Fanuc TP program (LS listing): 190220_hosenrohr_oV4.ls

/PROG  190220_hosenrohr_oV4
/ATTR
COMMENT	= "19-02-22 10:03:29";
PROG_SIZE	= 0;
DEFAULT_GROUP	= 1, 1, *, *, *;
/APPL
    ARC Welding Equipment: 1, *, *, *, *;
/MN
   1:  CALL HOME_ALL;
   1:  UFRAME_NUM = 1;
   1:  UTOOL_NUM = 3;
   1:  COL GUARD ADJUST 150;
   1:  ! -- Layer/Ebene 142 -- !;
   1:  PR[91] = PR[90];
   1:  PR[GP1:91,1] = PR[GP1:90,1] + -1.507;
   1:  PR[GP1:91,2] = PR[GP1:90,2] + 38.342;
   1:  PR[GP1:91,3] = PR[GP1:90,3] + 86.925;
   1:  !Sicherheitspunkt!;
   1:  PR[92] = PR[91];
   1:  PR[92] = PR[GP1:92,3] + 50;
   1:J PR[92];
   1:  !Schweissanfang anfahren!;
   1:L PR[91] R[100]mm/sec CNT100;
   1:  CALL LASER_DRAHT_START;
   1:  PR[GP1:91,1] = PR[GP1:90,1] + -7.188;
   1:  PR[GP1:91,2] = PR[GP1:90,2] + 40.092;
   1:L PR[91] R[100]mm/sec CNT100;
   1:  PR[GP1:91,1] = PR[GP1:90,1] + -15.510;
   1:  PR[GP1:91,2] = PR[GP1:90,2] + 40.391;
   1:L PR[91] R[100]mm/sec CNT100;
   1:  PR[GP1:91,1] = PR[GP1:90,1] + -22.386;
   1:  PR[GP1:91,2] = PR[GP1:90,2] + 40.265;
   1:L PR[91] R[100]mm/sec CNT100;
   1:  PR[GP1:91,1] = PR[GP1:90,1] + -29.270;
   1:  PR[GP1:91,2] = PR[GP1:90,2] + 38.008;
   1:L PR[91] R[100]mm/sec CNT100;
   1:  PR[GP1:91,1] = PR[GP1:90,1] + -36.534;
   1:  PR[GP1:91,2] = PR[GP1:90,2] + 35.327;
   1:L PR[91] R[100]mm/sec CNT100;
   1:  PR[GP1:91,1] = PR[GP1:90,1] + -41.379;
   1:  PR[GP1:91,2] = PR[GP1:90,2] + 31.493;
   1:L PR[91] R[100]mm/sec CNT100;
   1:  PR[GP1:91,1] = PR[GP1:90,1] + -47.922;
   1:  PR[GP1:91,2] = PR[GP1:90,2] + 26.092;
   1:L PR[91] R[100]mm/sec CNT100;
   1:  PR[GP1:91,1] = PR[GP1:90,1] + -50.649;
   1:  PR[GP1:91,2] = PR[GP1:90,2] + 21.582;
   1:L PR[91] R[100]mm/sec CNT100;
   1:  PR[GP1:91,1] = PR[GP1:90,1] + -55.262;
   1:  PR[GP1:91,2] = PR[GP1:90,2] + 13.777;
   1:L PR[91] R[100]mm/sec CNT100;
   1:  PR[GP1:91,1] = PR[GP1:90,1] + -56.985;
   1:  PR[GP1:91,2] = PR[GP1:90,2] + 4.269;
   1:L PR[91] R[100]mm/sec CNT100;
   1:  PR[GP1:91,1] = PR[GP1:90,1] + -57.684;
   1:  PR[GP1:91,2] = PR[GP1:90,2] + -0.066;
   1:L PR[91] R[100]mm/sec CNT100;
   1:  PR[GP1:91,1] = PR[GP1:90,1] + -56.617;
   1:  PR[GP1:91,2] = PR[GP1:90,2] + -5.926;
   1:L PR[91] R[100]mm/sec CNT100;
   1:  PR[GP1:91,1] = PR[GP1:90,1] + -56.104;
   1:  PR[GP1:91,2] = PR[GP1:90,2] + -9.354;
   1:L PR[91] R[100]mm/sec CNT100;
   1:  PR[GP1:91,1] = PR[GP1:90,1] + -55.261;
   1:  PR[GP1:91,2] = PR[GP1:90,2] + -13.923;
   1:L PR[91] R[100]mm/sec CNT100;
   1:  PR[GP1:91,1] = PR[GP1:90,1] + -50.646;
   1:  PR[GP1:91,2] = PR[GP1:90,2] + -21.730;
   1:L PR[91] R[100]mm/sec CNT100;
   1:  PR[GP1:91,1] = PR[GP1:90,1] + -47.919;
   1:  PR[GP1:91,2] = PR[GP1:90,2] + -26.240;
   1:L PR[91] R[100]mm/sec CNT100;
   1:  PR[GP1:91,1] = PR[GP1:90,1] + -41.373;
   1:  PR[GP1:91,2] = PR[GP1:90,2] + -31.640;
   1:L PR[91] R[100]mm/sec CNT100;
   1:  PR[GP1:91,1] = PR[GP1:90,1] + -36.528;
   1:  PR[GP1:91,2] = PR[GP1:90,2] + -35.474;
   1:L PR[91] R[100]mm/sec CNT100;
   1:  PR[GP1:91,1] = PR[GP1:90,1] + -29.263;
   1:  PR[GP1:91,2] = PR[GP1:90,2] + -38.152;
   1:L PR[91] R[100]mm/sec CNT100;
   1:  PR[GP1:91,1] = PR[GP1:90,1] + -22.379;
   1:  PR[GP1:91,2] = PR[GP1:90,2] + -40.411;
   1:L PR[91] R[100]mm/sec CNT100;
   1:  PR[GP1:91,1] = PR[GP1:90,1] + -15.502;
   1:  PR[GP1:91,2] = PR[GP1:90,2] + -40.533;
   1:L PR[91] R[100]mm/sec CNT100;
   1:  PR[GP1:91,1] = PR[GP1:90,1] + -7.183;
   1:  PR[GP1:91,2] = PR[GP1:90,2] + -40.236;
   1:L PR[91] R[100]mm/sec CNT100;
   1:  PR[GP1:91,1] = PR[GP1:90,1] + -1.509;
   1:  PR[GP1:91,2] = PR[GP1:90,2] + -38.475;
   1:L PR[91] R[100]mm/sec CNT100;
   1:  PR[GP1:91,1] = PR[GP1:90,1] + 1.722;
   1:  PR[GP1:91,2] = PR[GP1:90,2] + -38.474;
   1:L PR[91] R[100]mm/sec CNT100;
   1:  PR[GP1:91,1] = PR[GP1:90,1] + 7.396;
   1:  PR[GP1:91,2] = PR[GP1:90,2] + -40.236;
   1:L PR[91] R[100]mm/sec CNT100;
   1:  PR[GP1:91,1] = PR[GP1:90,1] + 15.715;
   1:  PR[GP1:91,2] = PR[GP1:90,2] + -40.532;
   1:L PR[91] R[100]mm/sec CNT100;
   1:  PR[GP1:91,1] = PR[GP1:90,1] + 22.592;
   1:  PR[GP1:91,2] = PR[GP1:90,2] + -40.411;
   1:L PR[91] R[100]mm/sec CNT100;
   1:  PR[GP1:91,1] = PR[GP1:90,1] + 29.475;
   1:  PR[GP1:91,2] = PR[GP1:90,2] + -38.153;
   1:L PR[91] R[100]mm/sec CNT100;
   1:  PR[GP1:91,1] = PR[GP1:90,1] + 36.742;
   1:  PR[GP1:91,2] = PR[GP1:90,2] + -35.476;
   1:L PR[91] R[100]mm/sec CNT100;
   1:  PR[GP1:91,1] = PR[GP1:90,1] + 41.585;
   1:  PR[GP1:91,2] = PR[GP1:90,2] + -31.641;
   1:L PR[91] R[100]mm/sec CNT100;
   1:  PR[GP1:91,1] = PR[GP1:90,1] + 48.132;
   1:  PR[GP1:91,2] = PR[GP1:90,2] + -26.235;
   1:L PR[91] R[100]mm/sec CNT100;
   1:  PR[GP1:91,1] = PR[GP1:90,1] + 50.859;
   1:  PR[GP1:91,2] = PR[GP1:90,2] + -21.727;
   1:L PR[91] R[100]mm/sec CNT100;
   1:  PR[GP1:91,1] = PR[GP1:90,1] + 55.474;
   1:  PR[GP1:91,2] = PR[GP1:90,2] + -13.938;
   1:L PR[91] R[100]mm/sec CNT100;
   1:  PR[GP1:91,1] = PR[GP1:90,1] + 57.199;
   1:  PR[GP1:91,2] = PR[GP1:90,2] + -4.414;
   1:L PR[91] R[100]mm/sec CNT100;
   1:  PR[GP1:91,1] = PR[GP1:90,1] + 57.897;
   1:  PR[GP1:91,2] = PR[GP1:90,2] + -0.078;
   1:L PR[91] R[100]mm/sec CNT100;
   1:  PR[GP1:91,1] = PR[GP1:90,1] + 56.831;
   1:  PR[GP1:91,2] = PR[GP1:90,2] + 5.789;
   1:L PR[91] R[100]mm/sec CNT100;
   1:  PR[GP1:91,1] = PR[GP1:90,1] + 56.318;
   1:  PR[GP1:91,2] = PR[GP1:90,2] + 9.220;
   1:L PR[91] R[100]mm/sec CNT100;
   1:  PR[GP1:91,1] = PR[GP1:90,1] + 55.475;
   1:  PR[GP1:91,2] = PR[GP1:90,2] + 13.790;
   1:L PR[91] R[100]mm/sec CNT100;
   1:  PR[GP1:91,1] = PR[GP1:90,1] + 50.862;
   1:  PR[GP1:91,2] = PR[GP1:90,2] + 21.580;
   1:L PR[91] R[100]mm/sec CNT100;
   1:  PR[GP1:91,1] = PR[GP1:90,1] + 48.135;
   1:  PR[GP1:91,2] = PR[GP1:90,2] + 26.088;
   1:L PR[91] R[100]mm/sec CNT100;
   1:  PR[GP1:91,1] = PR[GP1:90,1] + 41.591;
   1:  PR[GP1:91,2] = PR[GP1:90,2] + 31.494;
   1:L PR[91] R[100]mm/sec CNT100;
   1:  PR[GP1:91,1] = PR[GP1:90,1] + 36.747;
   1:  PR[GP1:91,2] = PR[GP1:90,2] + 35.329;
   1:L PR[91] R[100]mm/sec CNT100;
   1:  PR[GP1:91,1] = PR[GP1:90,1] + 29.483;
   1:  PR[GP1:91,2] = PR[GP1:90,2] + 38.008;
   1:L PR[91] R[100]mm/sec CNT100;
   1:  PR[GP1:91,1] = PR[GP1:90,1] + 22.599;
   1:  PR[GP1:91,2] = PR[GP1:90,2] + 40.266;
   1:L PR[91] R[100]mm/sec CNT100;
   1:  PR[GP1:91,1] = PR[GP1:90,1] + 15.722;
   1:  PR[GP1:91,2] = PR[GP1:90,2] + 40.390;
   1:L PR[91] R[100]mm/sec CNT100;
   1:  PR[GP1:91,1] = PR[GP1:90,1] + 7.401;
   1:  PR[GP1:91,2] = PR[GP1:90,2] + 40.092;
   1:L PR[91] R[100]mm/sec CNT100;
   1:  PR[GP1:91,1] = PR[GP1:90,1] + 1.720;
   1:  PR[GP1:91,2] = PR[GP1:90,2] + 38.342;
   1:L PR[91] R[100]mm/sec CNT100;
   1:  ! -- Layer/Ebene 143 -- !;
   1:  PR[91] = PR[90];
   1:  PR[GP1:91,1] = PR[GP1:90,1] + -1.481;
   1:  PR[GP1:91,2] = PR[GP1:90,2] + 38.516;
   1:  PR[GP1:91,3] = PR[GP1:90,3] + 87.535;
   1:L PR[91] R[100]mm/sec CNT100;
   1:  PR[GP1:91,1] = PR[GP1:90,1] + -6.890;
   1:  PR[GP1:91,2] = PR[GP1:90,2] + 40.181;
   1:L PR[91] R[100]mm/sec CNT100;
   1:  PR[GP1:91,1] = PR[GP1:90,1] + -15.548;
   1:  PR[GP1:91,2] = PR[GP1:90,2] + 40.491;
   1:L PR[91] R[100]mm/sec CNT100;
   1:  PR[GP1:91,1] = PR[GP1:90,1] + -22.125;
   1:  PR[GP1:91,2] = PR[GP1:90,2] + 40.371;
   1:L PR[91] R[100]mm/sec CNT100;
   1:  PR[GP1:91,1] = PR[GP1:90,1] + -29.339;
   1:  PR[GP1:91,2] = PR[GP1:90,2] + 38.006;
   1:L PR[91] R[100]mm/sec CNT100;
   1:  PR[GP1:91,1] = PR[GP1:90,1] + -36.313;
   1:  PR[GP1:91,2] = PR[GP1:90,2] + 35.432;
   1:L PR[91] R[100]mm/sec CNT100;
   1:  PR[GP1:91,1] = PR[GP1:90,1] + -41.439;
   1:  PR[GP1:91,2] = PR[GP1:90,2] + 31.376;
   1:L PR[91] R[100]mm/sec CNT100;
   1:  PR[GP1:91,1] = PR[GP1:90,1] + -47.738;
   1:  PR[GP1:91,2] = PR[GP1:90,2] + 26.177;
   1:L PR[91] R[100]mm/sec CNT100;
   1:  PR[GP1:91,1] = PR[GP1:90,1] + -50.656;
   1:  PR[GP1:91,2] = PR[GP1:90,2] + 21.350;
   1:L PR[91] R[100]mm/sec CNT100;
   1:  PR[GP1:91,1] = PR[GP1:90,1] + -55.103;
   1:  PR[GP1:91,2] = PR[GP1:90,2] + 13.825;
   1:L PR[91] R[100]mm/sec CNT100;
   1:  PR[GP1:91,1] = PR[GP1:90,1] + -56.765;
   1:  PR[GP1:91,2] = PR[GP1:90,2] + 4.657;
   1:L PR[91] R[100]mm/sec CNT100;
   1:  PR[GP1:91,1] = PR[GP1:90,1] + -57.526;
   1:  PR[GP1:91,2] = PR[GP1:90,2] + -0.066;
   1:L PR[91] R[100]mm/sec CNT100;
   1:  PR[GP1:91,1] = PR[GP1:90,1] + -56.569;
   1:  PR[GP1:91,2] = PR[GP1:90,2] + -5.328;
   1:L PR[91] R[100]mm/sec CNT100;
   1:  PR[GP1:91,1] = PR[GP1:90,1] + -56.014;
   1:  PR[GP1:91,2] = PR[GP1:90,2] + -9.028;
   1:L PR[91] R[100]mm/sec CNT100;
   1:  PR[GP1:91,1] = PR[GP1:90,1] + -55.103;
   1:  PR[GP1:91,2] = PR[GP1:90,2] + -13.970;
   1:L PR[91] R[100]mm/sec CNT100;
   1:  PR[GP1:91,1] = PR[GP1:90,1] + -50.653;
   1:  PR[GP1:91,2] = PR[GP1:90,2] + -21.498;
   1:L PR[91] R[100]mm/sec CNT100;
   1:  PR[GP1:91,1] = PR[GP1:90,1] + -47.735;
   1:  PR[GP1:91,2] = PR[GP1:90,2] + -26.324;
   1:L PR[91] R[100]mm/sec CNT100;
   1:  PR[GP1:91,1] = PR[GP1:90,1] + -41.433;
   1:  PR[GP1:91,2] = PR[GP1:90,2] + -31.523;
   1:L PR[91] R[100]mm/sec CNT100;
   1:  PR[GP1:91,1] = PR[GP1:90,1] + -36.307;
   1:  PR[GP1:91,2] = PR[GP1:90,2] + -35.579;
   1:L PR[91] R[100]mm/sec CNT100;
   1:  PR[GP1:91,1] = PR[GP1:90,1] + -29.332;
   1:  PR[GP1:91,2] = PR[GP1:90,2] + -38.150;
   1:L PR[91] R[100]mm/sec CNT100;
   1:  PR[GP1:91,1] = PR[GP1:90,1] + -22.118;
   1:  PR[GP1:91,2] = PR[GP1:90,2] + -40.517;
   1:L PR[91] R[100]mm/sec CNT100;
   1:  PR[GP1:91,1] = PR[GP1:90,1] + -15.540;
   1:  PR[GP1:91,2] = PR[GP1:90,2] + -40.633;
   1:L PR[91] R[100]mm/sec CNT100;
   1:  PR[GP1:91,1] = PR[GP1:90,1] + -6.886;
   1:  PR[GP1:91,2] = PR[GP1:90,2] + -40.325;
   1:L PR[91] R[100]mm/sec CNT100;
   1:  PR[GP1:91,1] = PR[GP1:90,1] + -1.483;
   1:  PR[GP1:91,2] = PR[GP1:90,2] + -38.649;
   1:L PR[91] R[100]mm/sec CNT100;
   1:  PR[GP1:91,1] = PR[GP1:90,1] + 1.697;
   1:  PR[GP1:91,2] = PR[GP1:90,2] + -38.648;
   1:L PR[91] R[100]mm/sec CNT100;
   1:  PR[GP1:91,1] = PR[GP1:90,1] + 7.100;
   1:  PR[GP1:91,2] = PR[GP1:90,2] + -40.325;
   1:L PR[91] R[100]mm/sec CNT100;
   1:  PR[GP1:91,1] = PR[GP1:90,1] + 15.753;
   1:  PR[GP1:91,2] = PR[GP1:90,2] + -40.633;
   1:L PR[91] R[100]mm/sec CNT100;
   1:  PR[GP1:91,1] = PR[GP1:90,1] + 22.331;
   1:  PR[GP1:91,2] = PR[GP1:90,2] + -40.517;
   1:L PR[91] R[100]mm/sec CNT100;
   1:  PR[GP1:91,1] = PR[GP1:90,1] + 29.544;
   1:  PR[GP1:91,2] = PR[GP1:90,2] + -38.150;
   1:L PR[91] R[100]mm/sec CNT100;
   1:  PR[GP1:91,1] = PR[GP1:90,1] + 36.520;
   1:  PR[GP1:91,2] = PR[GP1:90,2] + -35.581;
   1:L PR[91] R[100]mm/sec CNT100;
   1:  PR[GP1:91,1] = PR[GP1:90,1] + 41.646;
   1:  PR[GP1:91,2] = PR[GP1:90,2] + -31.523;
   1:L PR[91] R[100]mm/sec CNT100;
   1:  PR[GP1:91,1] = PR[GP1:90,1] + 47.948;
   1:  PR[GP1:91,2] = PR[GP1:90,2] + -26.319;
   1:L PR[91] R[100]mm/sec CNT100;
   1:  PR[GP1:91,1] = PR[GP1:90,1] + 50.866;
   1:  PR[GP1:91,2] = PR[GP1:90,2] + -21.495;
   1:L PR[91] R[100]mm/sec CNT100;
   1:  PR[GP1:91,1] = PR[GP1:90,1] + 55.315;
   1:  PR[GP1:91,2] = PR[GP1:90,2] + -13.984;
   1:L PR[91] R[100]mm/sec CNT100;
   1:  PR[GP1:91,1] = PR[GP1:90,1] + 56.979;
   1:  PR[GP1:91,2] = PR[GP1:90,2] + -4.802;
   1:L PR[91] R[100]mm/sec CNT100;
   1:  PR[GP1:91,1] = PR[GP1:90,1] + 57.740;
   1:  PR[GP1:91,2] = PR[GP1:90,2] + -0.078;
   1:L PR[91] R[100]mm/sec CNT100;
   1:  PR[GP1:91,1] = PR[GP1:90,1] + 56.782;
   1:  PR[GP1:91,2] = PR[GP1:90,2] + 5.190;
   1:L PR[91] R[100]mm/sec CNT100;
   1:  PR[GP1:91,1] = PR[GP1:90,1] + 56.228;
   1:  PR[GP1:91,2] = PR[GP1:90,2] + 8.895;
   1:L PR[91] R[100]mm/sec CNT100;
   1:  PR[GP1:91,1] = PR[GP1:90,1] + 55.317;
   1:  PR[GP1:91,2] = PR[GP1:90,2] + 13.837;
   1:L PR[91] R[100]mm/sec CNT100;
   1:  PR[GP1:91,1] = PR[GP1:90,1] + 50.869;
   1:  PR[GP1:91,2] = PR[GP1:90,2] + 21.347;
   1:L PR[91] R[100]mm/sec CNT100;
   1:  PR[GP1:91,1] = PR[GP1:90,1] + 47.951;
   1:  PR[GP1:91,2] = PR[GP1:90,2] + 26.172;
   1:L PR[91] R[100]mm/sec CNT100;
   1:  PR[GP1:91,1] = PR[GP1:90,1] + 41.651;
   1:  PR[GP1:91,2] = PR[GP1:90,2] + 31.377;
   1:L PR[91] R[100]mm/sec CNT100;
   1:  PR[GP1:91,1] = PR[GP1:90,1] + 36.526;
   1:  PR[GP1:91,2] = PR[GP1:90,2] + 35.434;
   1:L PR[91] R[100]mm/sec CNT100;
   1:  PR[GP1:91,1] = PR[GP1:90,1] + 29.552;
   1:  PR[GP1:91,2] = PR[GP1:90,2] + 38.006;
   1:L PR[91] R[100]mm/sec CNT100;
   1:  PR[GP1:91,1] = PR[GP1:90,1] + 22.338;
   1:  PR[GP1:91,2] = PR[GP1:90,2] + 40.372;
   1:L PR[91] R[100]mm/sec CNT100;
   1:  PR[GP1:91,1] = PR[GP1:90,1] + 15.761;
   1:  PR[GP1:91,2] = PR[GP1:90,2] + 40.491;
   1:L PR[91] R[100]mm/sec CNT100;
   1:  PR[GP1:91,1] = PR[GP1:90,1] + 7.103;
   1:  PR[GP1:91,2] = PR[GP1:90,2] + 40.181;
   1:L PR[91] R[100]mm/sec CNT100;
   1:  PR[GP1:91,1] = PR[GP1:90,1] + 1.695;
   1:  PR[GP1:91,2] = PR[GP1:90,2] + 38.515;
   1:L PR[91] R[100]mm/sec CNT100;
   1:  ! -- Layer/Ebene 144 -- !;
   1:  PR[91] = PR[90];
   1:  PR[GP1:91,1] = PR[GP1:90,1] + -1.456;
   1:  PR[GP1:91,2] = PR[GP1:90,2] + 38.689;
   1:  PR[GP1:91,3] = PR[GP1:90,3] + 88.145;
   1:L PR[91] R[100]mm/sec CNT100;
   1:  PR[GP1:91,1] = PR[GP1:90,1] + -6.592;
   1:  PR[GP1:91,2] = PR[GP1:90,2] + 40.270;
   1:L PR[91] R[100]mm/sec CNT100;
   1:  PR[GP1:91,1] = PR[GP1:90,1] + -15.586;
   1:  PR[GP1:91,2] = PR[GP1:90,2] + 40.592;
   1:L PR[91] R[100]mm/sec CNT100;
   1:  PR[GP1:91,1] = PR[GP1:90,1] + -21.864;
   1:  PR[GP1:91,2] = PR[GP1:90,2] + 40.477;
   1:L PR[91] R[100]mm/sec CNT100;
   1:  PR[GP1:91,1] = PR[GP1:90,1] + -29.408;
   1:  PR[GP1:91,2] = PR[GP1:90,2] + 38.003;
   1:L PR[91] R[100]mm/sec CNT100;
   1:  PR[GP1:91,1] = PR[GP1:90,1] + -36.091;
   1:  PR[GP1:91,2] = PR[GP1:90,2] + 35.537;
   1:L PR[91] R[100]mm/sec CNT100;
   1:  PR[GP1:91,1] = PR[GP1:90,1] + -41.499;
   1:  PR[GP1:91,2] = PR[GP1:90,2] + 31.258;
   1:L PR[91] R[100]mm/sec CNT100;
   1:  PR[GP1:91,1] = PR[GP1:90,1] + -47.553;
   1:  PR[GP1:91,2] = PR[GP1:90,2] + 26.261;
   1:L PR[91] R[100]mm/sec CNT100;
   1:  PR[GP1:91,1] = PR[GP1:90,1] + -50.663;
   1:  PR[GP1:91,2] = PR[GP1:90,2] + 21.117;
   1:L PR[91] R[100]mm/sec CNT100;
   1:  PR[GP1:91,1] = PR[GP1:90,1] + -54.945;
   1:  PR[GP1:91,2] = PR[GP1:90,2] + 13.872;
   1:L PR[91] R[100]mm/sec CNT100;
   1:  PR[GP1:91,1] = PR[GP1:90,1] + -56.545;
   1:  PR[GP1:91,2] = PR[GP1:90,2] + 5.045;
   1:L PR[91] R[100]mm/sec CNT100;
   1:  PR[GP1:91,1] = PR[GP1:90,1] + -57.369;
   1:  PR[GP1:91,2] = PR[GP1:90,2] + -0.066;
   1:L PR[91] R[100]mm/sec CNT100;
   1:  PR[GP1:91,1] = PR[GP1:90,1] + -56.520;
   1:  PR[GP1:91,2] = PR[GP1:90,2] + -4.730;
   1:L PR[91] R[100]mm/sec CNT100;
   1:  PR[GP1:91,1] = PR[GP1:90,1] + -55.925;
   1:  PR[GP1:91,2] = PR[GP1:90,2] + -8.703;
   1:L PR[91] R[100]mm/sec CNT100;
   1:  PR[GP1:91,1] = PR[GP1:90,1] + -54.944;
   1:  PR[GP1:91,2] = PR[GP1:90,2] + -14.017;
   1:L PR[91] R[100]mm/sec CNT100;
   1:  PR[GP1:91,1] = PR[GP1:90,1] + -50.660;
   1:  PR[GP1:91,2] = PR[GP1:90,2] + -21.265;
   1:L PR[91] R[100]mm/sec CNT100;
   1:  PR[GP1:91,1] = PR[GP1:90,1] + -47.550;
   1:  PR[GP1:91,2] = PR[GP1:90,2] + -26.408;
   1:L PR[91] R[100]mm/sec CNT100;
   1:  PR[GP1:91,1] = PR[GP1:90,1] + -41.493;
   1:  PR[GP1:91,2] = PR[GP1:90,2] + -31.405;
   1:L PR[91] R[100]mm/sec CNT100;
   1:  PR[GP1:91,1] = PR[GP1:90,1] + -36.086;
   1:  PR[GP1:91,2] = PR[GP1:90,2] + -35.684;
   1:L PR[91] R[100]mm/sec CNT100;
   1:  PR[GP1:91,1] = PR[GP1:90,1] + -29.401;
   1:  PR[GP1:91,2] = PR[GP1:90,2] + -38.148;
   1:L PR[91] R[100]mm/sec CNT100;
   1:  PR[GP1:91,1] = PR[GP1:90,1] + -21.857;
   1:  PR[GP1:91,2] = PR[GP1:90,2] + -40.623;
   1:L PR[91] R[100]mm/sec CNT100;
   1:  PR[GP1:91,1] = PR[GP1:90,1] + -15.579;
   1:  PR[GP1:91,2] = PR[GP1:90,2] + -40.734;
   1:L PR[91] R[100]mm/sec CNT100;
   1:  PR[GP1:91,1] = PR[GP1:90,1] + -6.589;
   1:  PR[GP1:91,2] = PR[GP1:90,2] + -40.414;
   1:L PR[91] R[100]mm/sec CNT100;
   1:  PR[GP1:91,1] = PR[GP1:90,1] + -1.458;
   1:  PR[GP1:91,2] = PR[GP1:90,2] + -38.822;
   1:L PR[91] R[100]mm/sec CNT100;
   1:  PR[GP1:91,1] = PR[GP1:90,1] + 1.671;
   1:L PR[91] R[100]mm/sec CNT100;
   1:  PR[GP1:91,1] = PR[GP1:90,1] + 6.803;
   1:  PR[GP1:91,2] = PR[GP1:90,2] + -40.413;
   1:L PR[91] R[100]mm/sec CNT100;
   1:  PR[GP1:91,1] = PR[GP1:90,1] + 15.792;
   1:  PR[GP1:91,2] = PR[GP1:90,2] + -40.734;
   1:L PR[91] R[100]mm/sec CNT100;
   1:  PR[GP1:91,1] = PR[GP1:90,1] + 22.071;
   1:  PR[GP1:91,2] = PR[GP1:90,2] + -40.623;
   1:L PR[91] R[100]mm/sec CNT100;
   1:  PR[GP1:91,1] = PR[GP1:90,1] + 29.613;
   1:  PR[GP1:91,2] = PR[GP1:90,2] + -38.148;
   1:L PR[91] R[100]mm/sec CNT100;
   1:  PR[GP1:91,1] = PR[GP1:90,1] + 36.299;
   1:  PR[GP1:91,2] = PR[GP1:90,2] + -35.685;
   1:L PR[91] R[100]mm/sec CNT100;
   1:  PR[GP1:91,1] = PR[GP1:90,1] + 41.706;
   1:  PR[GP1:91,2] = PR[GP1:90,2] + -31.405;
   1:L PR[91] R[100]mm/sec CNT100;
   1:  PR[GP1:91,1] = PR[GP1:90,1] + 47.763;
   1:  PR[GP1:91,2] = PR[GP1:90,2] + -26.403;
   1:L PR[91] R[100]mm/sec CNT100;
   1:  PR[GP1:91,1] = PR[GP1:90,1] + 50.873;
   1:  PR[GP1:91,2] = PR[GP1:90,2] + -21.262;
   1:L PR[91] R[100]mm/sec CNT100;
   1:  PR[GP1:91,1] = PR[GP1:90,1] + 55.157;
   1:  PR[GP1:91,2] = PR[GP1:90,2] + -14.031;
   1:L PR[91] R[100]mm/sec CNT100;
   1:  PR[GP1:91,1] = PR[GP1:90,1] + 56.758;
   1:  PR[GP1:91,2] = PR[GP1:90,2] + -5.190;
   1:L PR[91] R[100]mm/sec CNT100;
   1:  PR[GP1:91,1] = PR[GP1:90,1] + 57.582;
   1:  PR[GP1:91,2] = PR[GP1:90,2] + -0.078;
   1:L PR[91] R[100]mm/sec CNT100;
   1:  PR[GP1:91,1] = PR[GP1:90,1] + 56.733;
   1:  PR[GP1:91,2] = PR[GP1:90,2] + 4.591;
   1:L PR[91] R[100]mm/sec CNT100;
   1:  PR[GP1:91,1] = PR[GP1:90,1] + 56.139;
   1:  PR[GP1:91,2] = PR[GP1:90,2] + 8.569;
   1:L PR[91] R[100]mm/sec CNT100;
   1:  PR[GP1:91,1] = PR[GP1:90,1] + 55.158;
   1:  PR[GP1:91,2] = PR[GP1:90,2] + 13.884;
   1:L PR[91] R[100]mm/sec CNT100;
   1:  PR[GP1:91,1] = PR[GP1:90,1] + 50.876;
   1:  PR[GP1:91,2] = PR[GP1:90,2] + 21.115;
   1:L PR[91] R[100]mm/sec CNT100;
   1:  PR[GP1:91,1] = PR[GP1:90,1] + 47.766;
   1:  PR[GP1:91,2] = PR[GP1:90,2] + 26.256;
   1:L PR[91] R[100]mm/sec CNT100;
   1:  PR[GP1:91,1] = PR[GP1:90,1] + 41.711;
   1:  PR[GP1:91,2] = PR[GP1:90,2] + 31.259;
   1:L PR[91] R[100]mm/sec CNT100;
   1:  PR[GP1:91,1] = PR[GP1:90,1] + 36.304;
   1:  PR[GP1:91,2] = PR[GP1:90,2] + 35.539;
   1:L PR[91] R[100]mm/sec CNT100;
   1:  PR[GP1:91,1] = PR[GP1:90,1] + 29.620;
   1:  PR[GP1:91,2] = PR[GP1:90,2] + 38.004;
   1:L PR[91] R[100]mm/sec CNT100;
   1:  PR[GP1:91,1] = PR[GP1:90,1] + 22.077;
   1:  PR[GP1:91,2] = PR[GP1:90,2] + 40.478;
   1:L PR[91] R[100]mm/sec CNT100;
   1:  PR[GP1:91,1] = PR[GP1:90,1] + 15.799;
   1:  PR[GP1:91,2] = PR[GP1:90,2] + 40.591;
   1:L PR[91] R[100]mm/sec CNT100;
   1:  PR[GP1:91,1] = PR[GP1:90,1] + 6.806;
   1:  PR[GP1:91,2] = PR[GP1:90,2] + 40.269;
   1:L PR[91] R[100]mm/sec CNT100;
   1:  PR[GP1:91,1] = PR[GP1:90,1] + 1.670;
   1:  PR[GP1:91,2] = PR[GP1:90,2] + 38.688;
   1:L PR[91] R[100]mm/sec CNT100;
   1:  ! -- Layer/Ebene 145 -- !;
   1:  PR[91] = PR[90];
   1:  PR[GP1:91,1] = PR[GP1:90,1] + -1.431;
   1:  PR[GP1:91,2] = PR[GP1:90,2] + 38.862;
   1:  PR[GP1:91,3] = PR[GP1:90,3] + 88.755;
   1:L PR[91] R[100]mm/sec CNT100;
   1:  PR[GP1:91,1] = PR[GP1:90,1] + -6.295;
   1:  PR[GP1:91,2] = PR[GP1:90,2] + 40.358;
   1:L PR[91] R[100]mm/sec CNT100;
   1:  PR[GP1:91,1] = PR[GP1:90,1] + -15.624;
   1:  PR[GP1:91,2] = PR[GP1:90,2] + 40.693;
   1:L PR[91] R[100]mm/sec CNT100;
   1:  PR[GP1:91,1] = PR[GP1:90,1] + -21.602;
   1:  PR[GP1:91,2] = PR[GP1:90,2] + 40.584;
   1:L PR[91] R[100]mm/sec CNT100;
   1:  PR[GP1:91,1] = PR[GP1:90,1] + -29.476;
   1:  PR[GP1:91,2] = PR[GP1:90,2] + 38.002;
   1:L PR[91] R[100]mm/sec CNT100;
   1:  PR[GP1:91,1] = PR[GP1:90,1] + -35.870;
   1:  PR[GP1:91,2] = PR[GP1:90,2] + 35.642;
   1:L PR[91] R[100]mm/sec CNT100;
   1:  PR[GP1:91,1] = PR[GP1:90,1] + -41.558;
   1:  PR[GP1:91,2] = PR[GP1:90,2] + 31.140;
   1:L PR[91] R[100]mm/sec CNT100;
   1:  PR[GP1:91,1] = PR[GP1:90,1] + -47.368;
   1:  PR[GP1:91,2] = PR[GP1:90,2] + 26.345;
   1:L PR[91] R[100]mm/sec CNT100;
   1:  PR[GP1:91,1] = PR[GP1:90,1] + -50.670;
   1:  PR[GP1:91,2] = PR[GP1:90,2] + 20.884;
   1:L PR[91] R[100]mm/sec CNT100;
   1:  PR[GP1:91,1] = PR[GP1:90,1] + -54.786;
   1:  PR[GP1:91,2] = PR[GP1:90,2] + 13.919;
   1:L PR[91] R[100]mm/sec CNT100;
   1:  PR[GP1:91,1] = PR[GP1:90,1] + -56.324;
   1:  PR[GP1:91,2] = PR[GP1:90,2] + 5.433;
   1:L PR[91] R[100]mm/sec CNT100;
   1:  PR[GP1:91,1] = PR[GP1:90,1] + -57.211;
   1:  PR[GP1:91,2] = PR[GP1:90,2] + -0.066;
   1:L PR[91] R[100]mm/sec CNT100;
   1:  PR[GP1:91,1] = PR[GP1:90,1] + -56.471;
   1:  PR[GP1:91,2] = PR[GP1:90,2] + -4.131;
   1:L PR[91] R[100]mm/sec CNT100;
   1:  PR[GP1:91,1] = PR[GP1:90,1] + -55.835;
   1:  PR[GP1:91,2] = PR[GP1:90,2] + -8.377;
   1:L PR[91] R[100]mm/sec CNT100;
   1:  PR[GP1:91,1] = PR[GP1:90,1] + -54.786;
   1:  PR[GP1:91,2] = PR[GP1:90,2] + -14.064;
   1:L PR[91] R[100]mm/sec CNT100;
   1:  PR[GP1:91,1] = PR[GP1:90,1] + -50.667;
   1:  PR[GP1:91,2] = PR[GP1:90,2] + -21.032;
   1:L PR[91] R[100]mm/sec CNT100;
   1:  PR[GP1:91,1] = PR[GP1:90,1] + -47.366;
   1:  PR[GP1:91,2] = PR[GP1:90,2] + -26.492;
   1:L PR[91] R[100]mm/sec CNT100;
   1:  PR[GP1:91,1] = PR[GP1:90,1] + -41.553;
   1:  PR[GP1:91,2] = PR[GP1:90,2] + -31.287;
   1:L PR[91] R[100]mm/sec CNT100;
   1:  PR[GP1:91,1] = PR[GP1:90,1] + -35.865;
   1:  PR[GP1:91,2] = PR[GP1:90,2] + -35.789;
   1:L PR[91] R[100]mm/sec CNT100;
   1:  PR[GP1:91,1] = PR[GP1:90,1] + -29.469;
   1:  PR[GP1:91,2] = PR[GP1:90,2] + -38.146;
   1:L PR[91] R[100]mm/sec CNT100;
   1:  PR[GP1:91,1] = PR[GP1:90,1] + -21.596;
   1:  PR[GP1:91,2] = PR[GP1:90,2] + -40.729;
   1:L PR[91] R[100]mm/sec CNT100;
   1:  PR[GP1:91,1] = PR[GP1:90,1] + -15.618;
   1:  PR[GP1:91,2] = PR[GP1:90,2] + -40.835;
   1:L PR[91] R[100]mm/sec CNT100;
   1:  PR[GP1:91,1] = PR[GP1:90,1] + -6.292;
   1:  PR[GP1:91,2] = PR[GP1:90,2] + -40.502;
   1:L PR[91] R[100]mm/sec CNT100;
   1:  PR[GP1:91,1] = PR[GP1:90,1] + -1.433;
   1:  PR[GP1:91,2] = PR[GP1:90,2] + -38.996;
   1:L PR[91] R[100]mm/sec CNT100;
   1:  PR[GP1:91,1] = PR[GP1:90,1] + 1.646;
   1:  PR[GP1:91,2] = PR[GP1:90,2] + -38.995;
   1:L PR[91] R[100]mm/sec CNT100;
   1:  PR[GP1:91,1] = PR[GP1:90,1] + 6.506;
   1:  PR[GP1:91,2] = PR[GP1:90,2] + -40.502;
   1:L PR[91] R[100]mm/sec CNT100;
   1:  PR[GP1:91,1] = PR[GP1:90,1] + 15.831;
   1:  PR[GP1:91,2] = PR[GP1:90,2] + -40.834;
   1:L PR[91] R[100]mm/sec CNT100;
   1:  PR[GP1:91,1] = PR[GP1:90,1] + 21.810;
   1:  PR[GP1:91,2] = PR[GP1:90,2] + -40.729;
   1:L PR[91] R[100]mm/sec CNT100;
   1:  PR[GP1:91,1] = PR[GP1:90,1] + 29.682;
   1:  PR[GP1:91,2] = PR[GP1:90,2] + -38.146;
   1:L PR[91] R[100]mm/sec CNT100;
   1:  PR[GP1:91,1] = PR[GP1:90,1] + 36.078;
   1:  PR[GP1:91,2] = PR[GP1:90,2] + -35.790;
   1:L PR[91] R[100]mm/sec CNT100;
   1:  PR[GP1:91,1] = PR[GP1:90,1] + 41.766;
   1:  PR[GP1:91,2] = PR[GP1:90,2] + -31.287;
   1:L PR[91] R[100]mm/sec CNT100;
   1:  PR[GP1:91,1] = PR[GP1:90,1] + 47.579;
   1:  PR[GP1:91,2] = PR[GP1:90,2] + -26.487;
   1:L PR[91] R[100]mm/sec CNT100;
   1:  PR[GP1:91,1] = PR[GP1:90,1] + 50.880;
   1:  PR[GP1:91,2] = PR[GP1:90,2] + -21.029;
   1:L PR[91] R[100]mm/sec CNT100;
   1:  PR[GP1:91,1] = PR[GP1:90,1] + 54.998;
   1:  PR[GP1:91,2] = PR[GP1:90,2] + -14.078;
   1:L PR[91] R[100]mm/sec CNT100;
   1:  PR[GP1:91,1] = PR[GP1:90,1] + 56.538;
   1:  PR[GP1:91,2] = PR[GP1:90,2] + -5.579;
   1:L PR[91] R[100]mm/sec CNT100;
   1:  PR[GP1:91,1] = PR[GP1:90,1] + 57.424;
   1:  PR[GP1:91,2] = PR[GP1:90,2] + -0.078;
   1:L PR[91] R[100]mm/sec CNT100;
   1:  PR[GP1:91,1] = PR[GP1:90,1] + 56.684;
   1:  PR[GP1:91,2] = PR[GP1:90,2] + 3.992;
   1:L PR[91] R[100]mm/sec CNT100;
   1:  PR[GP1:91,1] = PR[GP1:90,1] + 56.049;
   1:  PR[GP1:91,2] = PR[GP1:90,2] + 8.243;
   1:L PR[91] R[100]mm/sec CNT100;
   1:  PR[GP1:91,1] = PR[GP1:90,1] + 55.000;
   1:  PR[GP1:91,2] = PR[GP1:90,2] + 13.931;
   1:L PR[91] R[100]mm/sec CNT100;
   1:  PR[GP1:91,1] = PR[GP1:90,1] + 50.883;
   1:  PR[GP1:91,2] = PR[GP1:90,2] + 20.882;
   1:L PR[91] R[100]mm/sec CNT100;
   1:  PR[GP1:91,1] = PR[GP1:90,1] + 47.581;
   1:  PR[GP1:91,2] = PR[GP1:90,2] + 26.340;
   1:L PR[91] R[100]mm/sec CNT100;
   1:  PR[GP1:91,1] = PR[GP1:90,1] + 41.771;
   1:  PR[GP1:91,2] = PR[GP1:90,2] + 31.141;
   1:L PR[91] R[100]mm/sec CNT100;
   1:  PR[GP1:91,1] = PR[GP1:90,1] + 36.083;
   1:  PR[GP1:91,2] = PR[GP1:90,2] + 35.643;
   1:L PR[91] R[100]mm/sec CNT100;
   1:  PR[GP1:91,1] = PR[GP1:90,1] + 29.689;
   1:  PR[GP1:91,2] = PR[GP1:90,2] + 38.002;
   1:L PR[91] R[100]mm/sec CNT100;
   1:  PR[GP1:91,1] = PR[GP1:90,1] + 21.816;
   1:  PR[GP1:91,2] = PR[GP1:90,2] + 40.584;
   1:L PR[91] R[100]mm/sec CNT100;
   1:  PR[GP1:91,1] = PR[GP1:90,1] + 15.837;
   1:  PR[GP1:91,2] = PR[GP1:90,2] + 40.692;
   1:L PR[91] R[100]mm/sec CNT100;
   1:  PR[GP1:91,1] = PR[GP1:90,1] + 6.508;
   1:  PR[GP1:91,2] = PR[GP1:90,2] + 40.358;
   1:L PR[91] R[100]mm/sec CNT100;
   1:  PR[GP1:91,1] = PR[GP1:90,1] + 1.645;
   1:  PR[GP1:91,2] = PR[GP1:90,2] + 38.861;
   1:L PR[91] R[100]mm/sec CNT100;
   1:  ! -- Layer/Ebene 146 -- !;
   1:  PR[91] = PR[90];
   1:  PR[GP1:91,1] = PR[GP1:90,1] + -1.406;
   1:  PR[GP1:91,2] = PR[GP1:90,2] + 39.035;
   1:  PR[GP1:91,3] = PR[GP1:90,3] + 89.365;
   1:L PR[91] R[100]mm/sec CNT100;
   1:  PR[GP1:91,1] = PR[GP1:90,1] + -5.997;
   1:  PR[GP1:91,2] = PR[GP1:90,2] + 40.447;
   1:L PR[91] R[100]mm/sec CNT100;
   1:  PR[GP1:91,1] = PR[GP1:90,1] + -15.662;
   1:  PR[GP1:91,2] = PR[GP1:90,2] + 40.793;
   1:L PR[91] R[100]mm/sec CNT100;
   1:  PR[GP1:91,1] = PR[GP1:90,1] + -21.341;
   1:  PR[GP1:91,2] = PR[GP1:90,2] + 40.690;
   1:L PR[91] R[100]mm/sec CNT100;
   1:  PR[GP1:91,1] = PR[GP1:90,1] + -29.544;
   1:  PR[GP1:91,2] = PR[GP1:90,2] + 38.000;
   1:L PR[91] R[100]mm/sec CNT100;
   1:  PR[GP1:91,1] = PR[GP1:90,1] + -35.648;
   1:  PR[GP1:91,2] = PR[GP1:90,2] + 35.747;
   1:L PR[91] R[100]mm/sec CNT100;
   1:  PR[GP1:91,1] = PR[GP1:90,1] + -41.618;
   1:  PR[GP1:91,2] = PR[GP1:90,2] + 31.023;
   1:L PR[91] R[100]mm/sec CNT100;
   1:  PR[GP1:91,1] = PR[GP1:90,1] + -47.184;
   1:  PR[GP1:91,2] = PR[GP1:90,2] + 26.429;
   1:L PR[91] R[100]mm/sec CNT100;
   1:  PR[GP1:91,1] = PR[GP1:90,1] + -50.677;
   1:  PR[GP1:91,2] = PR[GP1:90,2] + 20.652;
   1:L PR[91] R[100]mm/sec CNT100;
   1:  PR[GP1:91,1] = PR[GP1:90,1] + -54.628;
   1:  PR[GP1:91,2] = PR[GP1:90,2] + 13.966;
   1:L PR[91] R[100]mm/sec CNT100;
   1:  PR[GP1:91,1] = PR[GP1:90,1] + -56.104;
   1:  PR[GP1:91,2] = PR[GP1:90,2] + 5.821;
   1:L PR[91] R[100]mm/sec CNT100;
   1:  PR[GP1:91,1] = PR[GP1:90,1] + -57.053;
   1:  PR[GP1:91,2] = PR[GP1:90,2] + -0.066;
   1:L PR[91] R[100]mm/sec CNT100;
   1:  PR[GP1:91,1] = PR[GP1:90,1] + -56.422;
   1:  PR[GP1:91,2] = PR[GP1:90,2] + -3.533;
   1:L PR[91] R[100]mm/sec CNT100;
   1:  PR[GP1:91,1] = PR[GP1:90,1] + -55.745;
   1:  PR[GP1:91,2] = PR[GP1:90,2] + -8.052;
   1:L PR[91] R[100]mm/sec CNT100;
   1:  PR[GP1:91,1] = PR[GP1:90,1] + -54.627;
   1:  PR[GP1:91,2] = PR[GP1:90,2] + -14.111;
   1:L PR[91] R[100]mm/sec CNT100;
   1:  PR[GP1:91,1] = PR[GP1:90,1] + -50.674;
   1:  PR[GP1:91,2] = PR[GP1:90,2] + -20.799;
   1:L PR[91] R[100]mm/sec CNT100;
   1:  PR[GP1:91,1] = PR[GP1:90,1] + -47.181;
   1:  PR[GP1:91,2] = PR[GP1:90,2] + -26.576;
   1:L PR[91] R[100]mm/sec CNT100;
   1:  PR[GP1:91,1] = PR[GP1:90,1] + -41.613;
   1:  PR[GP1:91,2] = PR[GP1:90,2] + -31.169;
   1:L PR[91] R[100]mm/sec CNT100;
   1:  PR[GP1:91,1] = PR[GP1:90,1] + -35.644;
   1:  PR[GP1:91,2] = PR[GP1:90,2] + -35.893;
   1:L PR[91] R[100]mm/sec CNT100;
   1:  PR[GP1:91,1] = PR[GP1:90,1] + -29.538;
   1:  PR[GP1:91,2] = PR[GP1:90,2] + -38.144;
   1:L PR[91] R[100]mm/sec CNT100;
   1:  PR[GP1:91,1] = PR[GP1:90,1] + -21.335;
   1:  PR[GP1:91,2] = PR[GP1:90,2] + -40.835;
   1:L PR[91] R[100]mm/sec CNT100;
   1:  PR[GP1:91,1] = PR[GP1:90,1] + -15.656;
   1:  PR[GP1:91,2] = PR[GP1:90,2] + -40.936;
   1:L PR[91] R[100]mm/sec CNT100;
   1:  PR[GP1:91,1] = PR[GP1:90,1] + -5.995;
   1:  PR[GP1:91,2] = PR[GP1:90,2] + -40.591;
   1:L PR[91] R[100]mm/sec CNT100;
   1:  PR[GP1:91,1] = PR[GP1:90,1] + -1.408;
   1:  PR[GP1:91,2] = PR[GP1:90,2] + -39.170;
   1:L PR[91] R[100]mm/sec CNT100;
   1:  PR[GP1:91,1] = PR[GP1:90,1] + 1.621;
   1:  PR[GP1:91,2] = PR[GP1:90,2] + -39.169;
   1:L PR[91] R[100]mm/sec CNT100;
   1:  PR[GP1:91,1] = PR[GP1:90,1] + 6.209;
   1:  PR[GP1:91,2] = PR[GP1:90,2] + -40.591;
   1:L PR[91] R[100]mm/sec CNT100;
   1:  PR[GP1:91,1] = PR[GP1:90,1] + 15.870;
   1:  PR[GP1:91,2] = PR[GP1:90,2] + -40.935;
   1:L PR[91] R[100]mm/sec CNT100;
   1:  PR[GP1:91,1] = PR[GP1:90,1] + 21.549;
   1:  PR[GP1:91,2] = PR[GP1:90,2] + -40.835;
   1:L PR[91] R[100]mm/sec CNT100;
   1:  PR[GP1:91,1] = PR[GP1:90,1] + 29.751;
   1:  PR[GP1:91,2] = PR[GP1:90,2] + -38.144;
   1:L PR[91] R[100]mm/sec CNT100;
   1:  PR[GP1:91,1] = PR[GP1:90,1] + 35.857;
   1:  PR[GP1:91,2] = PR[GP1:90,2] + -35.895;
   1:L PR[91] R[100]mm/sec CNT100;
   1:  PR[GP1:91,1] = PR[GP1:90,1] + 41.826;
   1:  PR[GP1:91,2] = PR[GP1:90,2] + -31.169;
   1:L PR[91] R[100]mm/sec CNT100;
   1:  PR[GP1:91,1] = PR[GP1:90,1] + 47.394;
   1:  PR[GP1:91,2] = PR[GP1:90,2] + -26.571;
   1:L PR[91] R[100]mm/sec CNT100;
   1:  PR[GP1:91,1] = PR[GP1:90,1] + 50.887;
   1:  PR[GP1:91,2] = PR[GP1:90,2] + -20.797;
   1:L PR[91] R[100]mm/sec CNT100;
   1:  PR[GP1:91,1] = PR[GP1:90,1] + 54.840;
   1:  PR[GP1:91,2] = PR[GP1:90,2] + -14.125;
   1:L PR[91] R[100]mm/sec CNT100;
   1:  PR[GP1:91,1] = PR[GP1:90,1] + 56.318;
   1:  PR[GP1:91,2] = PR[GP1:90,2] + -5.967;
   1:L PR[91] R[100]mm/sec CNT100;
   1:  PR[GP1:91,1] = PR[GP1:90,1] + 57.266;
   1:  PR[GP1:91,2] = PR[GP1:90,2] + -0.078;
   1:L PR[91] R[100]mm/sec CNT100;
   1:  PR[GP1:91,1] = PR[GP1:90,1] + 56.636;
   1:  PR[GP1:91,2] = PR[GP1:90,2] + 3.393;
   1:L PR[91] R[100]mm/sec CNT100;
   1:  PR[GP1:91,1] = PR[GP1:90,1] + 55.959;
   1:  PR[GP1:91,2] = PR[GP1:90,2] + 7.917;
   1:L PR[91] R[100]mm/sec CNT100;
   1:  PR[GP1:91,1] = PR[GP1:90,1] + 54.841;
   1:  PR[GP1:91,2] = PR[GP1:90,2] + 13.978;
   1:L PR[91] R[100]mm/sec CNT100;
   1:  PR[GP1:91,1] = PR[GP1:90,1] + 50.890;
   1:  PR[GP1:91,2] = PR[GP1:90,2] + 20.650;
   1:L PR[91] R[100]mm/sec CNT100;
   1:  PR[GP1:91,1] = PR[GP1:90,1] + 47.397;
   1:  PR[GP1:91,2] = PR[GP1:90,2] + 26.425;
   1:L PR[91] R[100]mm/sec CNT100;
   1:  PR[GP1:91,1] = PR[GP1:90,1] + 41.831;
   1:  PR[GP1:91,2] = PR[GP1:90,2] + 31.023;
   1:L PR[91] R[100]mm/sec CNT100;
   1:  PR[GP1:91,1] = PR[GP1:90,1] + 35.861;
   1:  PR[GP1:91,2] = PR[GP1:90,2] + 35.748;
   1:L PR[91] R[100]mm/sec CNT100;
   1:  PR[GP1:91,1] = PR[GP1:90,1] + 29.757;
   1:  PR[GP1:91,2] = PR[GP1:90,2] + 38.000;
   1:L PR[91] R[100]mm/sec CNT100;
   1:  PR[GP1:91,1] = PR[GP1:90,1] + 21.554;
   1:  PR[GP1:91,2] = PR[GP1:90,2] + 40.690;
   1:L PR[91] R[100]mm/sec CNT100;
   1:  PR[GP1:91,1] = PR[GP1:90,1] + 15.876;
   1:  PR[GP1:91,2] = PR[GP1:90,2] + 40.793;
   1:L PR[91] R[100]mm/sec CNT100;
   1:  PR[GP1:91,1] = PR[GP1:90,1] + 6.211;
   1:  PR[GP1:91,2] = PR[GP1:90,2] + 40.447;
   1:L PR[91] R[100]mm/sec CNT100;
   1:  PR[GP1:91,1] = PR[GP1:90,1] + 1.620;
   1:  PR[GP1:91,2] = PR[GP1:90,2] + 39.035;
   1:L PR[91] R[100]mm/sec CNT100;
   1:  ! -- Layer/Ebene 147 -- !;
   1:  PR[91] = PR[90];
   1:  PR[GP1:91,1] = PR[GP1:90,1] + -1.380;
   1:  PR[GP1:91,2] = PR[GP1:90,2] + 39.208;
   1:  PR[GP1:91,3] = PR[GP1:90,3] + 89.975;
   1:L PR[91] R[100]mm/sec CNT100;
   1:  PR[GP1:91,1] = PR[GP1:90,1] + -5.699;
   1:  PR[GP1:91,2] = PR[GP1:90,2] + 40.535;
   1:L PR[91] R[100]mm/sec CNT100;
   1:  PR[GP1:91,1] = PR[GP1:90,1] + -15.700;
   1:  PR[GP1:91,2] = PR[GP1:90,2] + 40.894;
   1:L PR[91] R[100]mm/sec CNT100;
   1:  PR[GP1:91,1] = PR[GP1:90,1] + -21.079;
   1:  PR[GP1:91,2] = PR[GP1:90,2] + 40.796;
   1:L PR[91] R[100]mm/sec CNT100;
   1:  PR[GP1:91,1] = PR[GP1:90,1] + -29.613;
   1:  PR[GP1:91,2] = PR[GP1:90,2] + 37.998;
   1:L PR[91] R[100]mm/sec CNT100;
   1:  PR[GP1:91,1] = PR[GP1:90,1] + -35.427;
   1:  PR[GP1:91,2] = PR[GP1:90,2] + 35.852;
   1:L PR[91] R[100]mm/sec CNT100;
   1:  PR[GP1:91,1] = PR[GP1:90,1] + -41.678;
   1:  PR[GP1:91,2] = PR[GP1:90,2] + 30.905;
   1:L PR[91] R[100]mm/sec CNT100;
   1:  PR[GP1:91,1] = PR[GP1:90,1] + -46.999;
   1:  PR[GP1:91,2] = PR[GP1:90,2] + 26.513;
   1:L PR[91] R[100]mm/sec CNT100;
   1:  PR[GP1:91,1] = PR[GP1:90,1] + -50.684;
   1:  PR[GP1:91,2] = PR[GP1:90,2] + 20.419;
   1:L PR[91] R[100]mm/sec CNT100;
   1:  PR[GP1:91,1] = PR[GP1:90,1] + -54.469;
   1:  PR[GP1:91,2] = PR[GP1:90,2] + 14.013;
   1:L PR[91] R[100]mm/sec CNT100;
   1:  PR[GP1:91,1] = PR[GP1:90,1] + -55.884;
   1:  PR[GP1:91,2] = PR[GP1:90,2] + 6.209;
   1:L PR[91] R[100]mm/sec CNT100;
   1:  PR[GP1:91,1] = PR[GP1:90,1] + -56.895;
   1:  PR[GP1:91,2] = PR[GP1:90,2] + -0.066;
   1:L PR[91] R[100]mm/sec CNT100;
   1:  PR[GP1:91,1] = PR[GP1:90,1] + -56.373;
   1:  PR[GP1:91,2] = PR[GP1:90,2] + -2.934;
   1:L PR[91] R[100]mm/sec CNT100;
   1:  PR[GP1:91,1] = PR[GP1:90,1] + -55.656;
   1:  PR[GP1:91,2] = PR[GP1:90,2] + -7.726;
   1:L PR[91] R[100]mm/sec CNT100;
   1:  PR[GP1:91,1] = PR[GP1:90,1] + -54.469;
   1:  PR[GP1:91,2] = PR[GP1:90,2] + -14.158;
   1:L PR[91] R[100]mm/sec CNT100;
   1:  PR[GP1:91,1] = PR[GP1:90,1] + -50.681;
   1:  PR[GP1:91,2] = PR[GP1:90,2] + -20.566;
   1:L PR[91] R[100]mm/sec CNT100;
   1:  PR[GP1:91,1] = PR[GP1:90,1] + -46.997;
   1:  PR[GP1:91,2] = PR[GP1:90,2] + -26.660;
   1:L PR[91] R[100]mm/sec CNT100;
   1:  PR[GP1:91,1] = PR[GP1:90,1] + -41.673;
   1:  PR[GP1:91,2] = PR[GP1:90,2] + -31.051;
   1:L PR[91] R[100]mm/sec CNT100;
   1:  PR[GP1:91,1] = PR[GP1:90,1] + -35.422;
   1:  PR[GP1:91,2] = PR[GP1:90,2] + -35.998;
   1:L PR[91] R[100]mm/sec CNT100;
   1:  PR[GP1:91,1] = PR[GP1:90,1] + -29.607;
   1:  PR[GP1:91,2] = PR[GP1:90,2] + -38.142;
   1:L PR[91] R[100]mm/sec CNT100;
   1:  PR[GP1:91,1] = PR[GP1:90,1] + -21.075;
   1:  PR[GP1:91,2] = PR[GP1:90,2] + -40.941;
   1:L PR[91] R[100]mm/sec CNT100;
   1:  PR[GP1:91,1] = PR[GP1:90,1] + -15.695;
   1:  PR[GP1:91,2] = PR[GP1:90,2] + -41.036;
   1:L PR[91] R[100]mm/sec CNT100;
   1:  PR[GP1:91,1] = PR[GP1:90,1] + -5.698;
   1:  PR[GP1:91,2] = PR[GP1:90,2] + -40.680;
   1:L PR[91] R[100]mm/sec CNT100;
   1:  PR[GP1:91,1] = PR[GP1:90,1] + -1.382;
   1:  PR[GP1:91,2] = PR[GP1:90,2] + -39.343;
   1:L PR[91] R[100]mm/sec CNT100;
   1:  PR[GP1:91,1] = PR[GP1:90,1] + 1.596;
   1:L PR[91] R[100]mm/sec CNT100;
   1:  PR[GP1:91,1] = PR[GP1:90,1] + 5.913;
   1:  PR[GP1:91,2] = PR[GP1:90,2] + -40.680;
   1:L PR[91] R[100]mm/sec CNT100;
   1:  PR[GP1:91,1] = PR[GP1:90,1] + 15.909;
   1:  PR[GP1:91,2] = PR[GP1:90,2] + -41.036;
   1:L PR[91] R[100]mm/sec CNT100;
   1:  PR[GP1:91,1] = PR[GP1:90,1] + 21.288;
   1:  PR[GP1:91,2] = PR[GP1:90,2] + -40.941;
   1:L PR[91] R[100]mm/sec CNT100;
   1:  PR[GP1:91,1] = PR[GP1:90,1] + 29.820;
   1:  PR[GP1:91,2] = PR[GP1:90,2] + -38.142;
   1:L PR[91] R[100]mm/sec CNT100;
   1:  PR[GP1:91,1] = PR[GP1:90,1] + 35.636;
   1:  PR[GP1:91,2] = PR[GP1:90,2] + -36.000;
   1:L PR[91] R[100]mm/sec CNT100;
   1:  PR[GP1:91,1] = PR[GP1:90,1] + 41.886;
   1:  PR[GP1:91,2] = PR[GP1:90,2] + -31.051;
   1:L PR[91] R[100]mm/sec CNT100;
   1:  PR[GP1:91,1] = PR[GP1:90,1] + 47.210;
   1:  PR[GP1:91,2] = PR[GP1:90,2] + -26.655;
   1:L PR[91] R[100]mm/sec CNT100;
   1:  PR[GP1:91,1] = PR[GP1:90,1] + 50.894;
   1:  PR[GP1:91,2] = PR[GP1:90,2] + -20.564;
   1:L PR[91] R[100]mm/sec CNT100;
   1:  PR[GP1:91,1] = PR[GP1:90,1] + 54.682;
   1:  PR[GP1:91,2] = PR[GP1:90,2] + -14.171;
   1:L PR[91] R[100]mm/sec CNT100;
   1:  PR[GP1:91,1] = PR[GP1:90,1] + 56.097;
   1:  PR[GP1:91,2] = PR[GP1:90,2] + -6.355;
   1:L PR[91] R[100]mm/sec CNT100;
   1:  PR[GP1:91,1] = PR[GP1:90,1] + 57.109;
   1:  PR[GP1:91,2] = PR[GP1:90,2] + -0.078;
   1:L PR[91] R[100]mm/sec CNT100;
   1:  PR[GP1:91,1] = PR[GP1:90,1] + 56.587;
   1:  PR[GP1:91,2] = PR[GP1:90,2] + 2.794;
   1:L PR[91] R[100]mm/sec CNT100;
   1:  PR[GP1:91,1] = PR[GP1:90,1] + 55.870;
   1:  PR[GP1:91,2] = PR[GP1:90,2] + 7.591;
   1:L PR[91] R[100]mm/sec CNT100;
   1:  PR[GP1:91,1] = PR[GP1:90,1] + 54.683;
   1:  PR[GP1:91,2] = PR[GP1:90,2] + 14.025;
   1:L PR[91] R[100]mm/sec CNT100;
   1:  PR[GP1:91,1] = PR[GP1:90,1] + 50.897;
   1:  PR[GP1:91,2] = PR[GP1:90,2] + 20.417;
   1:L PR[91] R[100]mm/sec CNT100;
   1:  PR[GP1:91,1] = PR[GP1:90,1] + 47.212;
   1:  PR[GP1:91,2] = PR[GP1:90,2] + 26.509;
   1:L PR[91] R[100]mm/sec CNT100;
   1:  PR[GP1:91,1] = PR[GP1:90,1] + 41.891;
   1:  PR[GP1:91,2] = PR[GP1:90,2] + 30.905;
   1:L PR[91] R[100]mm/sec CNT100;
   1:  PR[GP1:91,1] = PR[GP1:90,1] + 35.640;
   1:  PR[GP1:91,2] = PR[GP1:90,2] + 35.853;
   1:L PR[91] R[100]mm/sec CNT100;
   1:  PR[GP1:91,1] = PR[GP1:90,1] + 29.826;
   1:  PR[GP1:91,2] = PR[GP1:90,2] + 37.998;
   1:L PR[91] R[100]mm/sec CNT100;
   1:  PR[GP1:91,1] = PR[GP1:90,1] + 21.293;
   1:  PR[GP1:91,2] = PR[GP1:90,2] + 40.796;
   1:L PR[91] R[100]mm/sec CNT100;
   1:  PR[GP1:91,1] = PR[GP1:90,1] + 15.914;
   1:  PR[GP1:91,2] = PR[GP1:90,2] + 40.894;
   1:L PR[91] R[100]mm/sec CNT100;
   1:  PR[GP1:91,1] = PR[GP1:90,1] + 5.913;
   1:  PR[GP1:91,2] = PR[GP1:90,2] + 40.535;
   1:L PR[91] R[100]mm/sec CNT100;
   1:  PR[GP1:91,1] = PR[GP1:90,1] + 1.594;
   1:  PR[GP1:91,2] = PR[GP1:90,2] + 39.208;
   1:L PR[91] R[100]mm/sec CNT100;
   1:  ! -- Layer/Ebene 148 -- !;
   1:  PR[91] = PR[90];
   1:  PR[GP1:91,1] = PR[GP1:90,1] + -1.355;
   1:  PR[GP1:91,2] = PR[GP1:90,2] + 39.381;
   1:  PR[GP1:91,3] = PR[GP1:90,3] + 90.585;
   1:L PR[91] R[100]mm/sec CNT100;
   1:  PR[GP1:91,1] = PR[GP1:90,1] + -5.402;
   1:  PR[GP1:91,2] = PR[GP1:90,2] + 40.624;
   1:L PR[91] R[100]mm/sec CNT100;
   1:  PR[GP1:91,1] = PR[GP1:90,1] + -15.739;
   1:  PR[GP1:91,2] = PR[GP1:90,2] + 40.995;
   1:L PR[91] R[100]mm/sec CNT100;
   1:  PR[GP1:91,1] = PR[GP1:90,1] + -20.818;
   1:  PR[GP1:91,2] = PR[GP1:90,2] + 40.902;
   1:L PR[91] R[100]mm/sec CNT100;
   1:  PR[GP1:91,1] = PR[GP1:90,1] + -29.681;
   1:  PR[GP1:91,2] = PR[GP1:90,2] + 37.996;
   1:L PR[91] R[100]mm/sec CNT100;
   1:  PR[GP1:91,1] = PR[GP1:90,1] + -35.205;
   1:  PR[GP1:91,2] = PR[GP1:90,2] + 35.957;
   1:L PR[91] R[100]mm/sec CNT100;
   1:  PR[GP1:91,1] = PR[GP1:90,1] + -41.738;
   1:  PR[GP1:91,2] = PR[GP1:90,2] + 30.787;
   1:L PR[91] R[100]mm/sec CNT100;
   1:  PR[GP1:91,1] = PR[GP1:90,1] + -46.814;
   1:  PR[GP1:91,2] = PR[GP1:90,2] + 26.597;
   1:L PR[91] R[100]mm/sec CNT100;
   1:  PR[GP1:91,1] = PR[GP1:90,1] + -50.691;
   1:  PR[GP1:91,2] = PR[GP1:90,2] + 20.186;
   1:L PR[91] R[100]mm/sec CNT100;
   1:  PR[GP1:91,1] = PR[GP1:90,1] + -54.311;
   1:  PR[GP1:91,2] = PR[GP1:90,2] + 14.061;
   1:L PR[91] R[100]mm/sec CNT100;
   1:  PR[GP1:91,1] = PR[GP1:90,1] + -55.664;
   1:  PR[GP1:91,2] = PR[GP1:90,2] + 6.598;
   1:L PR[91] R[100]mm/sec CNT100;
   1:  PR[GP1:91,1] = PR[GP1:90,1] + -56.738;
   1:  PR[GP1:91,2] = PR[GP1:90,2] + -0.066;
   1:L PR[91] R[100]mm/sec CNT100;
   1:  PR[GP1:91,1] = PR[GP1:90,1] + -56.324;
   1:  PR[GP1:91,2] = PR[GP1:90,2] + -2.336;
   1:L PR[91] R[100]mm/sec CNT100;
   1:  PR[GP1:91,1] = PR[GP1:90,1] + -55.566;
   1:  PR[GP1:91,2] = PR[GP1:90,2] + -7.401;
   1:L PR[91] R[100]mm/sec CNT100;
   1:  PR[GP1:91,1] = PR[GP1:90,1] + -54.310;
   1:  PR[GP1:91,2] = PR[GP1:90,2] + -14.205;
   1:L PR[91] R[100]mm/sec CNT100;
   1:  PR[GP1:91,1] = PR[GP1:90,1] + -50.688;
   1:  PR[GP1:91,2] = PR[GP1:90,2] + -20.333;
   1:L PR[91] R[100]mm/sec CNT100;
   1:  PR[GP1:91,1] = PR[GP1:90,1] + -46.812;
   1:  PR[GP1:91,2] = PR[GP1:90,2] + -26.744;
   1:L PR[91] R[100]mm/sec CNT100;
   1:  PR[GP1:91,1] = PR[GP1:90,1] + -41.733;
   1:  PR[GP1:91,2] = PR[GP1:90,2] + -30.933;
   1:L PR[91] R[100]mm/sec CNT100;
   1:  PR[GP1:91,1] = PR[GP1:90,1] + -35.201;
   1:  PR[GP1:91,2] = PR[GP1:90,2] + -36.103;
   1:L PR[91] R[100]mm/sec CNT100;
   1:  PR[GP1:91,1] = PR[GP1:90,1] + -29.676;
   1:  PR[GP1:91,2] = PR[GP1:90,2] + -38.140;
   1:L PR[91] R[100]mm/sec CNT100;
   1:  PR[GP1:91,1] = PR[GP1:90,1] + -20.814;
   1:  PR[GP1:91,2] = PR[GP1:90,2] + -41.047;
   1:L PR[91] R[100]mm/sec CNT100;
   1:  PR[GP1:91,1] = PR[GP1:90,1] + -15.734;
   1:  PR[GP1:91,2] = PR[GP1:90,2] + -41.137;
   1:L PR[91] R[100]mm/sec CNT100;
   1:  PR[GP1:91,1] = PR[GP1:90,1] + -5.401;
   1:  PR[GP1:91,2] = PR[GP1:90,2] + -40.769;
   1:L PR[91] R[100]mm/sec CNT100;
   1:  PR[GP1:91,1] = PR[GP1:90,1] + -1.357;
   1:  PR[GP1:91,2] = PR[GP1:90,2] + -39.517;
   1:L PR[91] R[100]mm/sec CNT100;
   1:  PR[GP1:91,1] = PR[GP1:90,1] + 1.571;
   1:L PR[91] R[100]mm/sec CNT100;
   1:  PR[GP1:91,1] = PR[GP1:90,1] + 5.616;
   1:  PR[GP1:91,2] = PR[GP1:90,2] + -40.768;
   1:L PR[91] R[100]mm/sec CNT100;
   1:  PR[GP1:91,1] = PR[GP1:90,1] + 15.948;
   1:  PR[GP1:91,2] = PR[GP1:90,2] + -41.137;
   1:L PR[91] R[100]mm/sec CNT100;
   1:  PR[GP1:91,1] = PR[GP1:90,1] + 21.028;
   1:  PR[GP1:91,2] = PR[GP1:90,2] + -41.047;
   1:L PR[91] R[100]mm/sec CNT100;
   1:  PR[GP1:91,1] = PR[GP1:90,1] + 29.889;
   1:  PR[GP1:91,2] = PR[GP1:90,2] + -38.140;
   1:L PR[91] R[100]mm/sec CNT100;
   1:  PR[GP1:91,1] = PR[GP1:90,1] + 35.415;
   1:  PR[GP1:91,2] = PR[GP1:90,2] + -36.104;
   1:L PR[91] R[100]mm/sec CNT100;
   1:  PR[GP1:91,1] = PR[GP1:90,1] + 41.946;
   1:  PR[GP1:91,2] = PR[GP1:90,2] + -30.934;
   1:L PR[91] R[100]mm/sec CNT100;
   1:  PR[GP1:91,1] = PR[GP1:90,1] + 47.025;
   1:  PR[GP1:91,2] = PR[GP1:90,2] + -26.740;
   1:L PR[91] R[100]mm/sec CNT100;
   1:  PR[GP1:91,1] = PR[GP1:90,1] + 50.901;
   1:  PR[GP1:91,2] = PR[GP1:90,2] + -20.331;
   1:L PR[91] R[100]mm/sec CNT100;
   1:  PR[GP1:91,1] = PR[GP1:90,1] + 54.523;
   1:  PR[GP1:91,2] = PR[GP1:90,2] + -14.218;
   1:L PR[91] R[100]mm/sec CNT100;
   1:  PR[GP1:91,1] = PR[GP1:90,1] + 55.877;
   1:  PR[GP1:91,2] = PR[GP1:90,2] + -6.743;
   1:L PR[91] R[100]mm/sec CNT100;
   1:  PR[GP1:91,1] = PR[GP1:90,1] + 56.951;
   1:  PR[GP1:91,2] = PR[GP1:90,2] + -0.078;
   1:L PR[91] R[100]mm/sec CNT100;
   1:  PR[GP1:91,1] = PR[GP1:90,1] + 56.538;
   1:  PR[GP1:91,2] = PR[GP1:90,2] + 2.195;
   1:L PR[91] R[100]mm/sec CNT100;
   1:  PR[GP1:91,1] = PR[GP1:90,1] + 55.780;
   1:  PR[GP1:91,2] = PR[GP1:90,2] + 7.265;
   1:L PR[91] R[100]mm/sec CNT100;
   1:  PR[GP1:91,1] = PR[GP1:90,1] + 54.524;
   1:  PR[GP1:91,2] = PR[GP1:90,2] + 14.072;
   1:L PR[91] R[100]mm/sec CNT100;
   1:  PR[GP1:91,1] = PR[GP1:90,1] + 50.904;
   1:  PR[GP1:91,2] = PR[GP1:90,2] + 20.185;
   1:L PR[91] R[100]mm/sec CNT100;
   1:  PR[GP1:91,1] = PR[GP1:90,1] + 47.027;
   1:  PR[GP1:91,2] = PR[GP1:90,2] + 26.593;
   1:L PR[91] R[100]mm/sec CNT100;
   1:  PR[GP1:91,1] = PR[GP1:90,1] + 41.950;
   1:  PR[GP1:91,2] = PR[GP1:90,2] + 30.788;
   1:L PR[91] R[100]mm/sec CNT100;
   1:  PR[GP1:91,1] = PR[GP1:90,1] + 35.418;
   1:  PR[GP1:91,2] = PR[GP1:90,2] + 35.958;
   1:L PR[91] R[100]mm/sec CNT100;
   1:  PR[GP1:91,1] = PR[GP1:90,1] + 29.894;
   1:  PR[GP1:91,2] = PR[GP1:90,2] + 37.995;
   1:L PR[91] R[100]mm/sec CNT100;
   1:  PR[GP1:91,1] = PR[GP1:90,1] + 21.032;
   1:  PR[GP1:91,2] = PR[GP1:90,2] + 40.902;
   1:L PR[91] R[100]mm/sec CNT100;
   1:  PR[GP1:91,1] = PR[GP1:90,1] + 15.952;
   1:  PR[GP1:91,2] = PR[GP1:90,2] + 40.994;
   1:L PR[91] R[100]mm/sec CNT100;
   1:  PR[GP1:91,1] = PR[GP1:90,1] + 5.616;
   1:  PR[GP1:91,2] = PR[GP1:90,2] + 40.624;
   1:L PR[91] R[100]mm/sec CNT100;
   1:  PR[GP1:91,1] = PR[GP1:90,1] + 1.569;
   1:  PR[GP1:91,2] = PR[GP1:90,2] + 39.381;
   1:L PR[91] R[100]mm/sec CNT100;
   1:  ! -- Layer/Ebene 149 -- !;
   1:  PR[91] = PR[90];
   1:  PR[GP1:91,1] = PR[GP1:90,1] + -1.330;
   1:  PR[GP1:91,2] = PR[GP1:90,2] + 39.555;
   1:  PR[GP1:91,3] = PR[GP1:90,3] + 91.195;
   1:L PR[91] R[100]mm/sec CNT100;
   1:  PR[GP1:91,1] = PR[GP1:90,1] + -5.104;
   1:  PR[GP1:91,2] = PR[GP1:90,2] + 40.713;
   1:L PR[91] R[100]mm/sec CNT100;
   1:  PR[GP1:91,1] = PR[GP1:90,1] + -15.777;
   1:  PR[GP1:91,2] = PR[GP1:90,2] + 41.095;
   1:L PR[91] R[100]mm/sec CNT100;
   1:  PR[GP1:91,1] = PR[GP1:90,1] + -20.557;
   1:  PR[GP1:91,2] = PR[GP1:90,2] + 41.008;
   1:L PR[91] R[100]mm/sec CNT100;
   1:  PR[GP1:91,1] = PR[GP1:90,1] + -29.749;
   1:  PR[GP1:91,2] = PR[GP1:90,2] + 37.994;
   1:L PR[91] R[100]mm/sec CNT100;
   1:  PR[GP1:91,1] = PR[GP1:90,1] + -34.983;
   1:  PR[GP1:91,2] = PR[GP1:90,2] + 36.062;
   1:L PR[91] R[100]mm/sec CNT100;
   1:  PR[GP1:91,1] = PR[GP1:90,1] + -41.798;
   1:  PR[GP1:91,2] = PR[GP1:90,2] + 30.670;
   1:L PR[91] R[100]mm/sec CNT100;
   1:  PR[GP1:91,1] = PR[GP1:90,1] + -46.630;
   1:  PR[GP1:91,2] = PR[GP1:90,2] + 26.682;
   1:L PR[91] R[100]mm/sec CNT100;
   1:  PR[GP1:91,1] = PR[GP1:90,1] + -50.698;
   1:  PR[GP1:91,2] = PR[GP1:90,2] + 19.953;
   1:L PR[91] R[100]mm/sec CNT100;
   1:  PR[GP1:91,1] = PR[GP1:90,1] + -54.152;
   1:  PR[GP1:91,2] = PR[GP1:90,2] + 14.108;
   1:L PR[91] R[100]mm/sec CNT100;
   1:  PR[GP1:91,1] = PR[GP1:90,1] + -55.443;
   1:  PR[GP1:91,2] = PR[GP1:90,2] + 6.986;
   1:L PR[91] R[100]mm/sec CNT100;
   1:  PR[GP1:91,1] = PR[GP1:90,1] + -56.580;
   1:  PR[GP1:91,2] = PR[GP1:90,2] + -0.066;
   1:L PR[91] R[100]mm/sec CNT100;
   1:  PR[GP1:91,1] = PR[GP1:90,1] + -56.275;
   1:  PR[GP1:91,2] = PR[GP1:90,2] + -1.738;
   1:L PR[91] R[100]mm/sec CNT100;
   1:  PR[GP1:91,1] = PR[GP1:90,1] + -55.476;
   1:  PR[GP1:91,2] = PR[GP1:90,2] + -7.075;
   1:L PR[91] R[100]mm/sec CNT100;
   1:  PR[GP1:91,1] = PR[GP1:90,1] + -54.152;
   1:  PR[GP1:91,2] = PR[GP1:90,2] + -14.253;
   1:L PR[91] R[100]mm/sec CNT100;
   1:  PR[GP1:91,1] = PR[GP1:90,1] + -50.695;
   1:  PR[GP1:91,2] = PR[GP1:90,2] + -20.100;
   1:L PR[91] R[100]mm/sec CNT100;
   1:  PR[GP1:91,1] = PR[GP1:90,1] + -46.628;
   1:  PR[GP1:91,2] = PR[GP1:90,2] + -26.828;
   1:L PR[91] R[100]mm/sec CNT100;
   1:  PR[GP1:91,1] = PR[GP1:90,1] + -41.793;
   1:  PR[GP1:91,2] = PR[GP1:90,2] + -30.816;
   1:L PR[91] R[100]mm/sec CNT100;
   1:  PR[GP1:91,1] = PR[GP1:90,1] + -34.980;
   1:  PR[GP1:91,2] = PR[GP1:90,2] + -36.208;
   1:L PR[91] R[100]mm/sec CNT100;
   1:  PR[GP1:91,1] = PR[GP1:90,1] + -29.745;
   1:  PR[GP1:91,2] = PR[GP1:90,2] + -38.138;
   1:L PR[91] R[100]mm/sec CNT100;
   1:  PR[GP1:91,1] = PR[GP1:90,1] + -20.553;
   1:  PR[GP1:91,2] = PR[GP1:90,2] + -41.153;
   1:L PR[91] R[100]mm/sec CNT100;
   1:  PR[GP1:91,1] = PR[GP1:90,1] + -15.773;
   1:  PR[GP1:91,2] = PR[GP1:90,2] + -41.238;
   1:L PR[91] R[100]mm/sec CNT100;
   1:  PR[GP1:91,1] = PR[GP1:90,1] + -5.105;
   1:  PR[GP1:91,2] = PR[GP1:90,2] + -40.857;
   1:L PR[91] R[100]mm/sec CNT100;
   1:  PR[GP1:91,1] = PR[GP1:90,1] + -1.332;
   1:  PR[GP1:91,2] = PR[GP1:90,2] + -39.691;
   1:L PR[91] R[100]mm/sec CNT100;
   1:  PR[GP1:91,1] = PR[GP1:90,1] + 1.546;
   1:  PR[GP1:91,2] = PR[GP1:90,2] + -39.690;
   1:L PR[91] R[100]mm/sec CNT100;
   1:  PR[GP1:91,1] = PR[GP1:90,1] + 5.319;
   1:  PR[GP1:91,2] = PR[GP1:90,2] + -40.857;
   1:L PR[91] R[100]mm/sec CNT100;
   1:  PR[GP1:91,1] = PR[GP1:90,1] + 15.986;
   1:  PR[GP1:91,2] = PR[GP1:90,2] + -41.237;
   1:L PR[91] R[100]mm/sec CNT100;
   1:  PR[GP1:91,1] = PR[GP1:90,1] + 20.767;
   1:  PR[GP1:91,2] = PR[GP1:90,2] + -41.153;
   1:L PR[91] R[100]mm/sec CNT100;
   1:  PR[GP1:91,1] = PR[GP1:90,1] + 29.958;
   1:  PR[GP1:91,2] = PR[GP1:90,2] + -38.138;
   1:L PR[91] R[100]mm/sec CNT100;
   1:  PR[GP1:91,1] = PR[GP1:90,1] + 35.194;
   1:  PR[GP1:91,2] = PR[GP1:90,2] + -36.209;
   1:L PR[91] R[100]mm/sec CNT100;
   1:  PR[GP1:91,1] = PR[GP1:90,1] + 42.006;
   1:  PR[GP1:91,2] = PR[GP1:90,2] + -30.816;
   1:L PR[91] R[100]mm/sec CNT100;
   1:  PR[GP1:91,1] = PR[GP1:90,1] + 46.841;
   1:  PR[GP1:91,2] = PR[GP1:90,2] + -26.824;
   1:L PR[91] R[100]mm/sec CNT100;
   1:  PR[GP1:91,1] = PR[GP1:90,1] + 50.909;
   1:  PR[GP1:91,2] = PR[GP1:90,2] + -20.099;
   1:L PR[91] R[100]mm/sec CNT100;
   1:  PR[GP1:91,1] = PR[GP1:90,1] + 54.365;
   1:  PR[GP1:91,2] = PR[GP1:90,2] + -14.265;
   1:L PR[91] R[100]mm/sec CNT100;
   1:  PR[GP1:91,1] = PR[GP1:90,1] + 55.657;
   1:  PR[GP1:91,2] = PR[GP1:90,2] + -7.131;
   1:L PR[91] R[100]mm/sec CNT100;
   1:  PR[GP1:91,1] = PR[GP1:90,1] + 56.793;
   1:  PR[GP1:91,2] = PR[GP1:90,2] + -0.078;
   1:L PR[91] R[100]mm/sec CNT100;
   1:  PR[GP1:91,1] = PR[GP1:90,1] + 56.489;
   1:  PR[GP1:91,2] = PR[GP1:90,2] + 1.596;
   1:L PR[91] R[100]mm/sec CNT100;
   1:  PR[GP1:91,1] = PR[GP1:90,1] + 55.690;
   1:  PR[GP1:91,2] = PR[GP1:90,2] + 6.939;
   1:L PR[91] R[100]mm/sec CNT100;
   1:  PR[GP1:91,1] = PR[GP1:90,1] + 54.366;
   1:  PR[GP1:91,2] = PR[GP1:90,2] + 14.119;
   1:L PR[91] R[100]mm/sec CNT100;
   1:  PR[GP1:91,1] = PR[GP1:90,1] + 50.911;
   1:  PR[GP1:91,2] = PR[GP1:90,2] + 19.952;
   1:L PR[91] R[100]mm/sec CNT100;
   1:  PR[GP1:91,1] = PR[GP1:90,1] + 46.843;
   1:  PR[GP1:91,2] = PR[GP1:90,2] + 26.677;
   1:L PR[91] R[100]mm/sec CNT100;
   1:  PR[GP1:91,1] = PR[GP1:90,1] + 42.010;
   1:  PR[GP1:91,2] = PR[GP1:90,2] + 30.670;
   1:L PR[91] R[100]mm/sec CNT100;
   1:  PR[GP1:91,1] = PR[GP1:90,1] + 35.197;
   1:  PR[GP1:91,2] = PR[GP1:90,2] + 36.063;
   1:L PR[91] R[100]mm/sec CNT100;
   1:  PR[GP1:91,1] = PR[GP1:90,1] + 29.963;
   1:  PR[GP1:91,2] = PR[GP1:90,2] + 37.993;
   1:L PR[91] R[100]mm/sec CNT100;
   1:  PR[GP1:91,1] = PR[GP1:90,1] + 20.771;
   1:  PR[GP1:91,2] = PR[GP1:90,2] + 41.008;
   1:L PR[91] R[100]mm/sec CNT100;
   1:  PR[GP1:91,1] = PR[GP1:90,1] + 15.991;
   1:  PR[GP1:91,2] = PR[GP1:90,2] + 41.095;
   1:L PR[91] R[100]mm/sec CNT100;
   1:  PR[GP1:91,1] = PR[GP1:90,1] + 5.318;
   1:  PR[GP1:91,2] = PR[GP1:90,2] + 40.712;
   1:L PR[91] R[100]mm/sec CNT100;
   1:  PR[GP1:91,1] = PR[GP1:90,1] + 1.544;
   1:  PR[GP1:91,2] = PR[GP1:90,2] + 39.554;
   1:L PR[91] R[100]mm/sec CNT100;
   1:  ! -- Layer/Ebene 150 -- !;
   1:  PR[91] = PR[90];
   1:  PR[GP1:91,1] = PR[GP1:90,1] + -1.304;
   1:  PR[GP1:91,2] = PR[GP1:90,2] + 39.728;
   1:  PR[GP1:91,3] = PR[GP1:90,3] + 91.805;
   1:L PR[91] R[100]mm/sec CNT100;
   1:  PR[GP1:91,1] = PR[GP1:90,1] + -4.806;
   1:  PR[GP1:91,2] = PR[GP1:90,2] + 40.801;
   1:L PR[91] R[100]mm/sec CNT100;
   1:  PR[GP1:91,1] = PR[GP1:90,1] + -15.815;
   1:  PR[GP1:91,2] = PR[GP1:90,2] + 41.196;
   1:L PR[91] R[100]mm/sec CNT100;
   1:  PR[GP1:91,1] = PR[GP1:90,1] + -20.295;
   1:  PR[GP1:91,2] = PR[GP1:90,2] + 41.114;
   1:L PR[91] R[100]mm/sec CNT100;
   1:  PR[GP1:91,1] = PR[GP1:90,1] + -29.818;
   1:  PR[GP1:91,2] = PR[GP1:90,2] + 37.992;
   1:L PR[91] R[100]mm/sec CNT100;
   1:  PR[GP1:91,1] = PR[GP1:90,1] + -34.762;
   1:  PR[GP1:91,2] = PR[GP1:90,2] + 36.167;
   1:L PR[91] R[100]mm/sec CNT100;
   1:  PR[GP1:91,1] = PR[GP1:90,1] + -41.858;
   1:  PR[GP1:91,2] = PR[GP1:90,2] + 30.552;
   1:L PR[91] R[100]mm/sec CNT100;
   1:  PR[GP1:91,1] = PR[GP1:90,1] + -46.445;
   1:  PR[GP1:91,2] = PR[GP1:90,2] + 26.766;
   1:L PR[91] R[100]mm/sec CNT100;
   1:  PR[GP1:91,1] = PR[GP1:90,1] + -50.705;
   1:  PR[GP1:91,2] = PR[GP1:90,2] + 19.721;
   1:L PR[91] R[100]mm/sec CNT100;
   1:  PR[GP1:91,1] = PR[GP1:90,1] + -53.994;
   1:  PR[GP1:91,2] = PR[GP1:90,2] + 14.155;
   1:L PR[91] R[100]mm/sec CNT100;
   1:  PR[GP1:91,1] = PR[GP1:90,1] + -55.223;
   1:  PR[GP1:91,2] = PR[GP1:90,2] + 7.374;
   1:L PR[91] R[100]mm/sec CNT100;
   1:  PR[GP1:91,1] = PR[GP1:90,1] + -56.422;
   1:  PR[GP1:91,2] = PR[GP1:90,2] + -0.066;
   1:L PR[91] R[100]mm/sec CNT100;
   1:  PR[GP1:91,1] = PR[GP1:90,1] + -56.227;
   1:  PR[GP1:91,2] = PR[GP1:90,2] + -1.139;
   1:L PR[91] R[100]mm/sec CNT100;
   1:  PR[GP1:91,1] = PR[GP1:90,1] + -55.387;
   1:  PR[GP1:91,2] = PR[GP1:90,2] + -6.749;
   1:L PR[91] R[100]mm/sec CNT100;
   1:  PR[GP1:91,1] = PR[GP1:90,1] + -53.993;
   1:  PR[GP1:91,2] = PR[GP1:90,2] + -14.300;
   1:L PR[91] R[100]mm/sec CNT100;
   1:  PR[GP1:91,1] = PR[GP1:90,1] + -50.702;
   1:  PR[GP1:91,2] = PR[GP1:90,2] + -19.867;
   1:L PR[91] R[100]mm/sec CNT100;
   1:  PR[GP1:91,1] = PR[GP1:90,1] + -46.443;
   1:  PR[GP1:91,2] = PR[GP1:90,2] + -26.912;
   1:L PR[91] R[100]mm/sec CNT100;
   1:  PR[GP1:91,1] = PR[GP1:90,1] + -41.853;
   1:  PR[GP1:91,2] = PR[GP1:90,2] + -30.698;
   1:L PR[91] R[100]mm/sec CNT100;
   1:  PR[GP1:91,1] = PR[GP1:90,1] + -34.759;
   1:  PR[GP1:91,2] = PR[GP1:90,2] + -36.313;
   1:L PR[91] R[100]mm/sec CNT100;
   1:  PR[GP1:91,1] = PR[GP1:90,1] + -29.814;
   1:  PR[GP1:91,2] = PR[GP1:90,2] + -38.136;
   1:L PR[91] R[100]mm/sec CNT100;
   1:  PR[GP1:91,1] = PR[GP1:90,1] + -20.292;
   1:  PR[GP1:91,2] = PR[GP1:90,2] + -41.259;
   1:L PR[91] R[100]mm/sec CNT100;
   1:  PR[GP1:91,1] = PR[GP1:90,1] + -15.811;
   1:  PR[GP1:91,2] = PR[GP1:90,2] + -41.339;
   1:L PR[91] R[100]mm/sec CNT100;
   1:  PR[GP1:91,1] = PR[GP1:90,1] + -4.808;
   1:  PR[GP1:91,2] = PR[GP1:90,2] + -40.946;
   1:L PR[91] R[100]mm/sec CNT100;
   1:  PR[GP1:91,1] = PR[GP1:90,1] + -1.306;
   1:  PR[GP1:91,2] = PR[GP1:90,2] + -39.864;
   1:L PR[91] R[100]mm/sec CNT100;
   1:  PR[GP1:91,1] = PR[GP1:90,1] + 1.521;
   1:L PR[91] R[100]mm/sec CNT100;
   1:  PR[GP1:91,1] = PR[GP1:90,1] + 5.022;
   1:  PR[GP1:91,2] = PR[GP1:90,2] + -40.946;
   1:L PR[91] R[100]mm/sec CNT100;
   1:  PR[GP1:91,1] = PR[GP1:90,1] + 16.025;
   1:  PR[GP1:91,2] = PR[GP1:90,2] + -41.338;
   1:L PR[91] R[100]mm/sec CNT100;
   1:  PR[GP1:91,1] = PR[GP1:90,1] + 20.506;
   1:  PR[GP1:91,2] = PR[GP1:90,2] + -41.259;
   1:L PR[91] R[100]mm/sec CNT100;
   1:  PR[GP1:91,1] = PR[GP1:90,1] + 30.027;
   1:  PR[GP1:91,2] = PR[GP1:90,2] + -38.136;
   1:L PR[91] R[100]mm/sec CNT100;
   1:  PR[GP1:91,1] = PR[GP1:90,1] + 34.973;
   1:  PR[GP1:91,2] = PR[GP1:90,2] + -36.314;
   1:L PR[91] R[100]mm/sec CNT100;
   1:  PR[GP1:91,1] = PR[GP1:90,1] + 42.067;
   1:  PR[GP1:91,2] = PR[GP1:90,2] + -30.697;
   1:L PR[91] R[100]mm/sec CNT100;
   1:  PR[GP1:91,1] = PR[GP1:90,1] + 46.656;
   1:  PR[GP1:91,2] = PR[GP1:90,2] + -26.908;
   1:L PR[91] R[100]mm/sec CNT100;
   1:  PR[GP1:91,1] = PR[GP1:90,1] + 50.916;
   1:  PR[GP1:91,2] = PR[GP1:90,2] + -19.866;
   1:L PR[91] R[100]mm/sec CNT100;
   1:  PR[GP1:91,1] = PR[GP1:90,1] + 54.206;
   1:  PR[GP1:91,2] = PR[GP1:90,2] + -14.312;
   1:L PR[91] R[100]mm/sec CNT100;
   1:  PR[GP1:91,1] = PR[GP1:90,1] + 55.437;
   1:  PR[GP1:91,2] = PR[GP1:90,2] + -7.520;
   1:L PR[91] R[100]mm/sec CNT100;
   1:  PR[GP1:91,1] = PR[GP1:90,1] + 56.635;
   1:  PR[GP1:91,2] = PR[GP1:90,2] + -0.078;
   1:L PR[91] R[100]mm/sec CNT100;
   1:  PR[GP1:91,1] = PR[GP1:90,1] + 56.440;
   1:  PR[GP1:91,2] = PR[GP1:90,2] + 0.997;
   1:L PR[91] R[100]mm/sec CNT100;
   1:  PR[GP1:91,1] = PR[GP1:90,1] + 55.600;
   1:  PR[GP1:91,2] = PR[GP1:90,2] + 6.613;
   1:L PR[91] R[100]mm/sec CNT100;
   1:  PR[GP1:91,1] = PR[GP1:90,1] + 54.207;
   1:  PR[GP1:91,2] = PR[GP1:90,2] + 14.165;
   1:L PR[91] R[100]mm/sec CNT100;
   1:  PR[GP1:91,1] = PR[GP1:90,1] + 50.918;
   1:  PR[GP1:91,2] = PR[GP1:90,2] + 19.720;
   1:L PR[91] R[100]mm/sec CNT100;
   1:  PR[GP1:91,1] = PR[GP1:90,1] + 46.658;
   1:  PR[GP1:91,2] = PR[GP1:90,2] + 26.761;
   1:L PR[91] R[100]mm/sec CNT100;
   1:  PR[GP1:91,1] = PR[GP1:90,1] + 42.070;
   1:  PR[GP1:91,2] = PR[GP1:90,2] + 30.552;
   1:L PR[91] R[100]mm/sec CNT100;
   1:  PR[GP1:91,1] = PR[GP1:90,1] + 34.976;
   1:  PR[GP1:91,2] = PR[GP1:90,2] + 36.168;
   1:L PR[91] R[100]mm/sec CNT100;
   1:  PR[GP1:91,1] = PR[GP1:90,1] + 30.031;
   1:  PR[GP1:91,2] = PR[GP1:90,2] + 37.991;
   1:L PR[91] R[100]mm/sec CNT100;
   1:  PR[GP1:91,1] = PR[GP1:90,1] + 20.509;
   1:  PR[GP1:91,2] = PR[GP1:90,2] + 41.115;
   1:L PR[91] R[100]mm/sec CNT100;
   1:  PR[GP1:91,1] = PR[GP1:90,1] + 16.029;
   1:  PR[GP1:91,2] = PR[GP1:90,2] + 41.196;
   1:L PR[91] R[100]mm/sec CNT100;
   1:  PR[GP1:91,1] = PR[GP1:90,1] + 5.021;
   1:  PR[GP1:91,2] = PR[GP1:90,2] + 40.801;
   1:L PR[91] R[100]mm/sec CNT100;
   1:  PR[GP1:91,1] = PR[GP1:90,1] + 1.519;
   1:  PR[GP1:91,2] = PR[GP1:90,2] + 39.727;
   1:L PR[91] R[100]mm/sec CNT100;
   1:  ! -- Layer/Ebene 151 -- !;
   1:  PR[91] = PR[90];
   1:  PR[GP1:91,1] = PR[GP1:90,1] + -1.279;
   1:  PR[GP1:91,2] = PR[GP1:90,2] + 39.901;
   1:  PR[GP1:91,3] = PR[GP1:90,3] + 92.415;
   1:L PR[91] R[100]mm/sec CNT100;
   1:  PR[GP1:91,1] = PR[GP1:90,1] + -4.509;
   1:  PR[GP1:91,2] = PR[GP1:90,2] + 40.890;
   1:L PR[91] R[100]mm/sec CNT100;
   1:  PR[GP1:91,1] = PR[GP1:90,1] + -15.853;
   1:  PR[GP1:91,2] = PR[GP1:90,2] + 41.297;
   1:L PR[91] R[100]mm/sec CNT100;
   1:  PR[GP1:91,1] = PR[GP1:90,1] + -20.034;
   1:  PR[GP1:91,2] = PR[GP1:90,2] + 41.221;
   1:L PR[91] R[100]mm/sec CNT100;
   1:  PR[GP1:91,1] = PR[GP1:90,1] + -29.886;
   1:  PR[GP1:91,2] = PR[GP1:90,2] + 37.990;
   1:L PR[91] R[100]mm/sec CNT100;
   1:  PR[GP1:91,1] = PR[GP1:90,1] + -34.540;
   1:  PR[GP1:91,2] = PR[GP1:90,2] + 36.272;
   1:L PR[91] R[100]mm/sec CNT100;
   1:  PR[GP1:91,1] = PR[GP1:90,1] + -41.917;
   1:  PR[GP1:91,2] = PR[GP1:90,2] + 30.434;
   1:L PR[91] R[100]mm/sec CNT100;
   1:  PR[GP1:91,1] = PR[GP1:90,1] + -46.260;
   1:  PR[GP1:91,2] = PR[GP1:90,2] + 26.850;
   1:L PR[91] R[100]mm/sec CNT100;
   1:  PR[GP1:91,1] = PR[GP1:90,1] + -50.712;
   1:  PR[GP1:91,2] = PR[GP1:90,2] + 19.488;
   1:L PR[91] R[100]mm/sec CNT100;
   1:  PR[GP1:91,1] = PR[GP1:90,1] + -53.835;
   1:  PR[GP1:91,2] = PR[GP1:90,2] + 14.202;
   1:L PR[91] R[100]mm/sec CNT100;
   1:  PR[GP1:91,1] = PR[GP1:90,1] + -55.003;
   1:  PR[GP1:91,2] = PR[GP1:90,2] + 7.762;
   1:L PR[91] R[100]mm/sec CNT100;
   1:  PR[GP1:91,1] = PR[GP1:90,1] + -56.264;
   1:  PR[GP1:91,2] = PR[GP1:90,2] + -0.066;
   1:L PR[91] R[100]mm/sec CNT100;
   1:  PR[GP1:91,1] = PR[GP1:90,1] + -56.178;
   1:  PR[GP1:91,2] = PR[GP1:90,2] + -0.541;
   1:L PR[91] R[100]mm/sec CNT100;
   1:  PR[GP1:91,1] = PR[GP1:90,1] + -55.297;
   1:  PR[GP1:91,2] = PR[GP1:90,2] + -6.424;
   1:L PR[91] R[100]mm/sec CNT100;
   1:  PR[GP1:91,1] = PR[GP1:90,1] + -53.835;
   1:  PR[GP1:91,2] = PR[GP1:90,2] + -14.347;
   1:L PR[91] R[100]mm/sec CNT100;
   1:  PR[GP1:91,1] = PR[GP1:90,1] + -50.709;
   1:  PR[GP1:91,2] = PR[GP1:90,2] + -19.634;
   1:L PR[91] R[100]mm/sec CNT100;
   1:  PR[GP1:91,1] = PR[GP1:90,1] + -46.258;
   1:  PR[GP1:91,2] = PR[GP1:90,2] + -26.996;
   1:L PR[91] R[100]mm/sec CNT100;
   1:  PR[GP1:91,1] = PR[GP1:90,1] + -41.914;
   1:  PR[GP1:91,2] = PR[GP1:90,2] + -30.580;
   1:L PR[91] R[100]mm/sec CNT100;
   1:  PR[GP1:91,1] = PR[GP1:90,1] + -34.538;
   1:  PR[GP1:91,2] = PR[GP1:90,2] + -36.417;
   1:L PR[91] R[100]mm/sec CNT100;
   1:  PR[GP1:91,1] = PR[GP1:90,1] + -29.882;
   1:  PR[GP1:91,2] = PR[GP1:90,2] + -38.133;
   1:L PR[91] R[100]mm/sec CNT100;
   1:  PR[GP1:91,1] = PR[GP1:90,1] + -20.031;
   1:  PR[GP1:91,2] = PR[GP1:90,2] + -41.365;
   1:L PR[91] R[100]mm/sec CNT100;
   1:  PR[GP1:91,1] = PR[GP1:90,1] + -15.850;
   1:  PR[GP1:91,2] = PR[GP1:90,2] + -41.439;
   1:L PR[91] R[100]mm/sec CNT100;
   1:  PR[GP1:91,1] = PR[GP1:90,1] + -4.511;
   1:  PR[GP1:91,2] = PR[GP1:90,2] + -41.035;
   1:L PR[91] R[100]mm/sec CNT100;
   1:  PR[GP1:91,1] = PR[GP1:90,1] + -1.281;
   1:  PR[GP1:91,2] = PR[GP1:90,2] + -40.038;
   1:L PR[91] R[100]mm/sec CNT100;
   1:  PR[GP1:91,1] = PR[GP1:90,1] + 1.495;
   1:L PR[91] R[100]mm/sec CNT100;
   1:  PR[GP1:91,1] = PR[GP1:90,1] + 4.725;
   1:  PR[GP1:91,2] = PR[GP1:90,2] + -41.035;
   1:L PR[91] R[100]mm/sec CNT100;
   1:  PR[GP1:91,1] = PR[GP1:90,1] + 16.064;
   1:  PR[GP1:91,2] = PR[GP1:90,2] + -41.439;
   1:L PR[91] R[100]mm/sec CNT100;
   1:  PR[GP1:91,1] = PR[GP1:90,1] + 20.245;
   1:  PR[GP1:91,2] = PR[GP1:90,2] + -41.365;
   1:L PR[91] R[100]mm/sec CNT100;
   1:  PR[GP1:91,1] = PR[GP1:90,1] + 30.096;
   1:  PR[GP1:91,2] = PR[GP1:90,2] + -38.133;
   1:L PR[91] R[100]mm/sec CNT100;
   1:  PR[GP1:91,1] = PR[GP1:90,1] + 34.751;
   1:  PR[GP1:91,2] = PR[GP1:90,2] + -36.418;
   1:L PR[91] R[100]mm/sec CNT100;
   1:  PR[GP1:91,1] = PR[GP1:90,1] + 42.127;
   1:  PR[GP1:91,2] = PR[GP1:90,2] + -30.580;
   1:L PR[91] R[100]mm/sec CNT100;
   1:  PR[GP1:91,1] = PR[GP1:90,1] + 46.472;
   1:  PR[GP1:91,2] = PR[GP1:90,2] + -26.992;
   1:L PR[91] R[100]mm/sec CNT100;
   1:  PR[GP1:91,1] = PR[GP1:90,1] + 50.923;
   1:  PR[GP1:91,2] = PR[GP1:90,2] + -19.633;
   1:L PR[91] R[100]mm/sec CNT100;
   1:  PR[GP1:91,1] = PR[GP1:90,1] + 54.048;
   1:  PR[GP1:91,2] = PR[GP1:90,2] + -14.358;
   1:L PR[91] R[100]mm/sec CNT100;
   1:  PR[GP1:91,1] = PR[GP1:90,1] + 55.216;
   1:  PR[GP1:91,2] = PR[GP1:90,2] + -7.908;
   1:L PR[91] R[100]mm/sec CNT100;
   1:  PR[GP1:91,1] = PR[GP1:90,1] + 56.478;
   1:  PR[GP1:91,2] = PR[GP1:90,2] + -0.078;
   1:L PR[91] R[100]mm/sec CNT100;
   1:  PR[GP1:91,1] = PR[GP1:90,1] + 56.391;
   1:  PR[GP1:91,2] = PR[GP1:90,2] + 0.398;
   1:L PR[91] R[100]mm/sec CNT100;
   1:  PR[GP1:91,1] = PR[GP1:90,1] + 55.511;
   1:  PR[GP1:91,2] = PR[GP1:90,2] + 6.287;
   1:L PR[91] R[100]mm/sec CNT100;
   1:  PR[GP1:91,1] = PR[GP1:90,1] + 54.049;
   1:  PR[GP1:91,2] = PR[GP1:90,2] + 14.212;
   1:L PR[91] R[100]mm/sec CNT100;
   1:  PR[GP1:91,1] = PR[GP1:90,1] + 50.925;
   1:  PR[GP1:91,2] = PR[GP1:90,2] + 19.487;
   1:L PR[91] R[100]mm/sec CNT100;
   1:  PR[GP1:91,1] = PR[GP1:90,1] + 46.474;
   1:  PR[GP1:91,2] = PR[GP1:90,2] + 26.846;
   1:L PR[91] R[100]mm/sec CNT100;
   1:  PR[GP1:91,1] = PR[GP1:90,1] + 42.130;
   1:  PR[GP1:91,2] = PR[GP1:90,2] + 30.434;
   1:L PR[91] R[100]mm/sec CNT100;
   1:  PR[GP1:91,1] = PR[GP1:90,1] + 34.754;
   1:  PR[GP1:91,2] = PR[GP1:90,2] + 36.273;
   1:L PR[91] R[100]mm/sec CNT100;
   1:  PR[GP1:91,1] = PR[GP1:90,1] + 30.100;
   1:  PR[GP1:91,2] = PR[GP1:90,2] + 37.989;
   1:L PR[91] R[100]mm/sec CNT100;
   1:  PR[GP1:91,1] = PR[GP1:90,1] + 20.248;
   1:  PR[GP1:91,2] = PR[GP1:90,2] + 41.221;
   1:L PR[91] R[100]mm/sec CNT100;
   1:  PR[GP1:91,1] = PR[GP1:90,1] + 16.067;
   1:  PR[GP1:91,2] = PR[GP1:90,2] + 41.296;
   1:L PR[91] R[100]mm/sec CNT100;
   1:  PR[GP1:91,1] = PR[GP1:90,1] + 4.723;
   1:  PR[GP1:91,2] = PR[GP1:90,2] + 40.890;
   1:L PR[91] R[100]mm/sec CNT100;
   1:  PR[GP1:91,1] = PR[GP1:90,1] + 1.494;
   1:  PR[GP1:91,2] = PR[GP1:90,2] + 39.901;
   1:L PR[91] R[100]mm/sec CNT100;
   1:  ! -- Layer/Ebene 152 -- !;
   1:  PR[91] = PR[90];
   1:  PR[GP1:91,1] = PR[GP1:90,1] + -1.254;
   1:  PR[GP1:91,2] = PR[GP1:90,2] + 40.074;
   1:  PR[GP1:91,3] = PR[GP1:90,3] + 93.025;
   1:L PR[91] R[100]mm/sec CNT100;
   1:  PR[GP1:91,1] = PR[GP1:90,1] + -4.211;
   1:  PR[GP1:91,2] = PR[GP1:90,2] + 40.979;
   1:L PR[91] R[100]mm/sec CNT100;
   1:  PR[GP1:91,1] = PR[GP1:90,1] + -15.891;
   1:  PR[GP1:91,2] = PR[GP1:90,2] + 41.398;
   1:L PR[91] R[100]mm/sec CNT100;
   1:  PR[GP1:91,1] = PR[GP1:90,1] + -19.773;
   1:  PR[GP1:91,2] = PR[GP1:90,2] + 41.327;
   1:L PR[91] R[100]mm/sec CNT100;
   1:  PR[GP1:91,1] = PR[GP1:90,1] + -29.955;
   1:  PR[GP1:91,2] = PR[GP1:90,2] + 37.988;
   1:L PR[91] R[100]mm/sec CNT100;
   1:  PR[GP1:91,1] = PR[GP1:90,1] + -34.319;
   1:  PR[GP1:91,2] = PR[GP1:90,2] + 36.377;
   1:L PR[91] R[100]mm/sec CNT100;
   1:  PR[GP1:91,1] = PR[GP1:90,1] + -41.977;
   1:  PR[GP1:91,2] = PR[GP1:90,2] + 30.317;
   1:L PR[91] R[100]mm/sec CNT100;
   1:  PR[GP1:91,1] = PR[GP1:90,1] + -46.076;
   1:  PR[GP1:91,2] = PR[GP1:90,2] + 26.934;
   1:L PR[91] R[100]mm/sec CNT100;
   1:  PR[GP1:91,1] = PR[GP1:90,1] + -50.718;
   1:  PR[GP1:91,2] = PR[GP1:90,2] + 19.255;
   1:L PR[91] R[100]mm/sec CNT100;
   1:  PR[GP1:91,1] = PR[GP1:90,1] + -53.677;
   1:  PR[GP1:91,2] = PR[GP1:90,2] + 14.249;
   1:L PR[91] R[100]mm/sec CNT100;
   1:  PR[GP1:91,1] = PR[GP1:90,1] + -54.782;
   1:  PR[GP1:91,2] = PR[GP1:90,2] + 8.150;
   1:L PR[91] R[100]mm/sec CNT100;
   1:  PR[GP1:91,1] = PR[GP1:90,1] + -56.109;
   1:  PR[GP1:91,2] = PR[GP1:90,2] + -0.075;
   1:L PR[91] R[100]mm/sec CNT100;
   1:  PR[GP1:91,1] = PR[GP1:90,1] + -55.207;
   1:  PR[GP1:91,2] = PR[GP1:90,2] + -6.098;
   1:L PR[91] R[100]mm/sec CNT100;
   1:  PR[GP1:91,1] = PR[GP1:90,1] + -53.677;
   1:  PR[GP1:91,2] = PR[GP1:90,2] + -14.394;
   1:L PR[91] R[100]mm/sec CNT100;
   1:  PR[GP1:91,1] = PR[GP1:90,1] + -50.716;
   1:  PR[GP1:91,2] = PR[GP1:90,2] + -19.401;
   1:L PR[91] R[100]mm/sec CNT100;
   1:  PR[GP1:91,1] = PR[GP1:90,1] + -46.074;
   1:  PR[GP1:91,2] = PR[GP1:90,2] + -27.080;
   1:L PR[91] R[100]mm/sec CNT100;
   1:  PR[GP1:91,1] = PR[GP1:90,1] + -41.974;
   1:  PR[GP1:91,2] = PR[GP1:90,2] + -30.462;
   1:L PR[91] R[100]mm/sec CNT100;
   1:  PR[GP1:91,1] = PR[GP1:90,1] + -34.316;
   1:  PR[GP1:91,2] = PR[GP1:90,2] + -36.522;
   1:L PR[91] R[100]mm/sec CNT100;
   1:  PR[GP1:91,1] = PR[GP1:90,1] + -29.951;
   1:  PR[GP1:91,2] = PR[GP1:90,2] + -38.131;
   1:L PR[91] R[100]mm/sec CNT100;
   1:  PR[GP1:91,1] = PR[GP1:90,1] + -19.770;
   1:  PR[GP1:91,2] = PR[GP1:90,2] + -41.471;
   1:L PR[91] R[100]mm/sec CNT100;
   1:  PR[GP1:91,1] = PR[GP1:90,1] + -15.889;
   1:  PR[GP1:91,2] = PR[GP1:90,2] + -41.540;
   1:L PR[91] R[100]mm/sec CNT100;
   1:  PR[GP1:91,1] = PR[GP1:90,1] + -4.214;
   1:  PR[GP1:91,2] = PR[GP1:90,2] + -41.124;
   1:L PR[91] R[100]mm/sec CNT100;
   1:  PR[GP1:91,1] = PR[GP1:90,1] + -1.255;
   1:  PR[GP1:91,2] = PR[GP1:90,2] + -40.212;
   1:L PR[91] R[100]mm/sec CNT100;
   1:  PR[GP1:91,1] = PR[GP1:90,1] + 1.470;
   1:  PR[GP1:91,2] = PR[GP1:90,2] + -40.211;
   1:L PR[91] R[100]mm/sec CNT100;
   1:  PR[GP1:91,1] = PR[GP1:90,1] + 4.428;
   1:  PR[GP1:91,2] = PR[GP1:90,2] + -41.124;
   1:L PR[91] R[100]mm/sec CNT100;
   1:  PR[GP1:91,1] = PR[GP1:90,1] + 16.103;
   1:  PR[GP1:91,2] = PR[GP1:90,2] + -41.540;
   1:L PR[91] R[100]mm/sec CNT100;
   1:  PR[GP1:91,1] = PR[GP1:90,1] + 19.985;
   1:  PR[GP1:91,2] = PR[GP1:90,2] + -41.471;
   1:L PR[91] R[100]mm/sec CNT100;
   1:  PR[GP1:91,1] = PR[GP1:90,1] + 30.165;
   1:  PR[GP1:91,2] = PR[GP1:90,2] + -38.131;
   1:L PR[91] R[100]mm/sec CNT100;
   1:  PR[GP1:91,1] = PR[GP1:90,1] + 34.530;
   1:  PR[GP1:91,2] = PR[GP1:90,2] + -36.523;
   1:L PR[91] R[100]mm/sec CNT100;
   1:  PR[GP1:91,1] = PR[GP1:90,1] + 42.187;
   1:  PR[GP1:91,2] = PR[GP1:90,2] + -30.461;
   1:L PR[91] R[100]mm/sec CNT100;
   1:  PR[GP1:91,1] = PR[GP1:90,1] + 46.287;
   1:  PR[GP1:91,2] = PR[GP1:90,2] + -27.076;
   1:L PR[91] R[100]mm/sec CNT100;
   1:  PR[GP1:91,1] = PR[GP1:90,1] + 50.930;
   1:  PR[GP1:91,2] = PR[GP1:90,2] + -19.401;
   1:L PR[91] R[100]mm/sec CNT100;
   1:  PR[GP1:91,1] = PR[GP1:90,1] + 53.889;
   1:  PR[GP1:91,2] = PR[GP1:90,2] + -14.405;
   1:L PR[91] R[100]mm/sec CNT100;
   1:  PR[GP1:91,1] = PR[GP1:90,1] + 54.996;
   1:  PR[GP1:91,2] = PR[GP1:90,2] + -8.296;
   1:L PR[91] R[100]mm/sec CNT100;
   1:  PR[GP1:91,1] = PR[GP1:90,1] + 56.322;
   1:  PR[GP1:91,2] = PR[GP1:90,2] + -0.069;
   1:L PR[91] R[100]mm/sec CNT100;
   1:  PR[GP1:91,1] = PR[GP1:90,1] + 55.421;
   1:  PR[GP1:91,2] = PR[GP1:90,2] + 5.961;
   1:L PR[91] R[100]mm/sec CNT100;
   1:  PR[GP1:91,1] = PR[GP1:90,1] + 53.890;
   1:  PR[GP1:91,2] = PR[GP1:90,2] + 14.259;
   1:L PR[91] R[100]mm/sec CNT100;
   1:  PR[GP1:91,1] = PR[GP1:90,1] + 50.932;
   1:  PR[GP1:91,2] = PR[GP1:90,2] + 19.255;
   1:L PR[91] R[100]mm/sec CNT100;
   1:  PR[GP1:91,1] = PR[GP1:90,1] + 46.289;
   1:  PR[GP1:91,2] = PR[GP1:90,2] + 26.930;
   1:L PR[91] R[100]mm/sec CNT100;
   1:  PR[GP1:91,1] = PR[GP1:90,1] + 42.190;
   1:  PR[GP1:91,2] = PR[GP1:90,2] + 30.316;
   1:L PR[91] R[100]mm/sec CNT100;
   1:  PR[GP1:91,1] = PR[GP1:90,1] + 34.533;
   1:  PR[GP1:91,2] = PR[GP1:90,2] + 36.378;
   1:L PR[91] R[100]mm/sec CNT100;
   1:  PR[GP1:91,1] = PR[GP1:90,1] + 30.168;
   1:  PR[GP1:91,2] = PR[GP1:90,2] + 37.987;
   1:L PR[91] R[100]mm/sec CNT100;
   1:  PR[GP1:91,1] = PR[GP1:90,1] + 19.987;
   1:  PR[GP1:91,2] = PR[GP1:90,2] + 41.327;
   1:L PR[91] R[100]mm/sec CNT100;
   1:  PR[GP1:91,1] = PR[GP1:90,1] + 16.106;
   1:  PR[GP1:91,2] = PR[GP1:90,2] + 41.397;
   1:L PR[91] R[100]mm/sec CNT100;
   1:  PR[GP1:91,1] = PR[GP1:90,1] + 4.426;
   1:  PR[GP1:91,2] = PR[GP1:90,2] + 40.978;
   1:L PR[91] R[100]mm/sec CNT100;
   1:  PR[GP1:91,1] = PR[GP1:90,1] + 1.469;
   1:  PR[GP1:91,2] = PR[GP1:90,2] + 40.074;
   1:L PR[91] R[100]mm/sec CNT100;
   1:  ! -- Layer/Ebene 153 -- !;
   1:  PR[91] = PR[90];
   1:  PR[GP1:91,1] = PR[GP1:90,1] + -1.228;
   1:  PR[GP1:91,2] = PR[GP1:90,2] + 40.247;
   1:  PR[GP1:91,3] = PR[GP1:90,3] + 93.635;
   1:L PR[91] R[100]mm/sec CNT100;
   1:  PR[GP1:91,1] = PR[GP1:90,1] + -3.913;
   1:  PR[GP1:91,2] = PR[GP1:90,2] + 41.067;
   1:L PR[91] R[100]mm/sec CNT100;
   1:  PR[GP1:91,1] = PR[GP1:90,1] + -15.930;
   1:  PR[GP1:91,2] = PR[GP1:90,2] + 41.498;
   1:L PR[91] R[100]mm/sec CNT100;
   1:  PR[GP1:91,1] = PR[GP1:90,1] + -19.511;
   1:  PR[GP1:91,2] = PR[GP1:90,2] + 41.433;
   1:L PR[91] R[100]mm/sec CNT100;
   1:  PR[GP1:91,1] = PR[GP1:90,1] + -30.023;
   1:  PR[GP1:91,2] = PR[GP1:90,2] + 37.985;
   1:L PR[91] R[100]mm/sec CNT100;
   1:  PR[GP1:91,1] = PR[GP1:90,1] + -34.097;
   1:  PR[GP1:91,2] = PR[GP1:90,2] + 36.482;
   1:L PR[91] R[100]mm/sec CNT100;
   1:  PR[GP1:91,1] = PR[GP1:90,1] + -42.037;
   1:  PR[GP1:91,2] = PR[GP1:90,2] + 30.199;
   1:L PR[91] R[100]mm/sec CNT100;
   1:  PR[GP1:91,1] = PR[GP1:90,1] + -45.891;
   1:  PR[GP1:91,2] = PR[GP1:90,2] + 27.018;
   1:L PR[91] R[100]mm/sec CNT100;
   1:  PR[GP1:91,1] = PR[GP1:90,1] + -50.725;
   1:  PR[GP1:91,2] = PR[GP1:90,2] + 19.022;
   1:L PR[91] R[100]mm/sec CNT100;
   1:  PR[GP1:91,1] = PR[GP1:90,1] + -53.518;
   1:  PR[GP1:91,2] = PR[GP1:90,2] + 14.297;
   1:L PR[91] R[100]mm/sec CNT100;
   1:  PR[GP1:91,1] = PR[GP1:90,1] + -54.562;
   1:  PR[GP1:91,2] = PR[GP1:90,2] + 8.538;
   1:L PR[91] R[100]mm/sec CNT100;
   1:  PR[GP1:91,1] = PR[GP1:90,1] + -55.823;
   1:  PR[GP1:91,2] = PR[GP1:90,2] + 0.713;
   1:L PR[91] R[100]mm/sec CNT100;
   1:  PR[GP1:91,1] = PR[GP1:90,1] + -55.970;
   1:  PR[GP1:91,2] = PR[GP1:90,2] + -0.082;
   1:L PR[91] R[100]mm/sec CNT100;
   1:  PR[GP1:91,1] = PR[GP1:90,1] + -55.117;
   1:  PR[GP1:91,2] = PR[GP1:90,2] + -5.773;
   1:L PR[91] R[100]mm/sec CNT100;
   1:  PR[GP1:91,1] = PR[GP1:90,1] + -53.518;
   1:  PR[GP1:91,2] = PR[GP1:90,2] + -14.441;
   1:L PR[91] R[100]mm/sec CNT100;
   1:  PR[GP1:91,1] = PR[GP1:90,1] + -50.723;
   1:  PR[GP1:91,2] = PR[GP1:90,2] + -19.168;
   1:L PR[91] R[100]mm/sec CNT100;
   1:  PR[GP1:91,1] = PR[GP1:90,1] + -45.889;
   1:  PR[GP1:91,2] = PR[GP1:90,2] + -27.164;
   1:L PR[91] R[100]mm/sec CNT100;
   1:  PR[GP1:91,1] = PR[GP1:90,1] + -42.034;
   1:  PR[GP1:91,2] = PR[GP1:90,2] + -30.344;
   1:L PR[91] R[100]mm/sec CNT100;
   1:  PR[GP1:91,1] = PR[GP1:90,1] + -34.095;
   1:  PR[GP1:91,2] = PR[GP1:90,2] + -36.627;
   1:L PR[91] R[100]mm/sec CNT100;
   1:  PR[GP1:91,1] = PR[GP1:90,1] + -30.020;
   1:  PR[GP1:91,2] = PR[GP1:90,2] + -38.129;
   1:L PR[91] R[100]mm/sec CNT100;
   1:  PR[GP1:91,1] = PR[GP1:90,1] + -19.509;
   1:  PR[GP1:91,2] = PR[GP1:90,2] + -41.577;
   1:L PR[91] R[100]mm/sec CNT100;
   1:  PR[GP1:91,1] = PR[GP1:90,1] + -15.927;
   1:  PR[GP1:91,2] = PR[GP1:90,2] + -41.641;
   1:L PR[91] R[100]mm/sec CNT100;
   1:  PR[GP1:91,1] = PR[GP1:90,1] + -3.917;
   1:  PR[GP1:91,2] = PR[GP1:90,2] + -41.213;
   1:L PR[91] R[100]mm/sec CNT100;
   1:  PR[GP1:91,1] = PR[GP1:90,1] + -1.230;
   1:  PR[GP1:91,2] = PR[GP1:90,2] + -40.385;
   1:L PR[91] R[100]mm/sec CNT100;
   1:  PR[GP1:91,1] = PR[GP1:90,1] + 1.445;
   1:L PR[91] R[100]mm/sec CNT100;
   1:  PR[GP1:91,1] = PR[GP1:90,1] + 4.132;
   1:  PR[GP1:91,2] = PR[GP1:90,2] + -41.212;
   1:L PR[91] R[100]mm/sec CNT100;
   1:  PR[GP1:91,1] = PR[GP1:90,1] + 16.142;
   1:  PR[GP1:91,2] = PR[GP1:90,2] + -41.640;
   1:L PR[91] R[100]mm/sec CNT100;
   1:  PR[GP1:91,1] = PR[GP1:90,1] + 19.724;
   1:  PR[GP1:91,2] = PR[GP1:90,2] + -41.577;
   1:L PR[91] R[100]mm/sec CNT100;
   1:  PR[GP1:91,1] = PR[GP1:90,1] + 30.233;
   1:  PR[GP1:91,2] = PR[GP1:90,2] + -38.129;
   1:L PR[91] R[100]mm/sec CNT100;
   1:  PR[GP1:91,1] = PR[GP1:90,1] + 34.309;
   1:  PR[GP1:91,2] = PR[GP1:90,2] + -36.628;
   1:L PR[91] R[100]mm/sec CNT100;
   1:  PR[GP1:91,1] = PR[GP1:90,1] + 42.247;
   1:  PR[GP1:91,2] = PR[GP1:90,2] + -30.344;
   1:L PR[91] R[100]mm/sec CNT100;
   1:  PR[GP1:91,1] = PR[GP1:90,1] + 46.103;
   1:  PR[GP1:91,2] = PR[GP1:90,2] + -27.160;
   1:L PR[91] R[100]mm/sec CNT100;
   1:  PR[GP1:91,1] = PR[GP1:90,1] + 50.937;
   1:  PR[GP1:91,2] = PR[GP1:90,2] + -19.168;
   1:L PR[91] R[100]mm/sec CNT100;
   1:  PR[GP1:91,1] = PR[GP1:90,1] + 53.731;
   1:  PR[GP1:91,2] = PR[GP1:90,2] + -14.452;
   1:L PR[91] R[100]mm/sec CNT100;
   1:  PR[GP1:91,1] = PR[GP1:90,1] + 54.776;
   1:  PR[GP1:91,2] = PR[GP1:90,2] + -8.684;
   1:L PR[91] R[100]mm/sec CNT100;
   1:  PR[GP1:91,1] = PR[GP1:90,1] + 56.037;
   1:  PR[GP1:91,2] = PR[GP1:90,2] + -0.857;
   1:L PR[91] R[100]mm/sec CNT100;
   1:  PR[GP1:91,1] = PR[GP1:90,1] + 56.183;
   1:  PR[GP1:91,2] = PR[GP1:90,2] + -0.062;
   1:L PR[91] R[100]mm/sec CNT100;
   1:  PR[GP1:91,1] = PR[GP1:90,1] + 55.331;
   1:  PR[GP1:91,2] = PR[GP1:90,2] + 5.635;
   1:L PR[91] R[100]mm/sec CNT100;
   1:  PR[GP1:91,1] = PR[GP1:90,1] + 53.732;
   1:  PR[GP1:91,2] = PR[GP1:90,2] + 14.306;
   1:L PR[91] R[100]mm/sec CNT100;
   1:  PR[GP1:91,1] = PR[GP1:90,1] + 50.939;
   1:  PR[GP1:91,2] = PR[GP1:90,2] + 19.022;
   1:L PR[91] R[100]mm/sec CNT100;
   1:  PR[GP1:91,1] = PR[GP1:90,1] + 46.104;
   1:  PR[GP1:91,2] = PR[GP1:90,2] + 27.014;
   1:L PR[91] R[100]mm/sec CNT100;
   1:  PR[GP1:91,1] = PR[GP1:90,1] + 42.250;
   1:  PR[GP1:91,2] = PR[GP1:90,2] + 30.199;
   1:L PR[91] R[100]mm/sec CNT100;
   1:  PR[GP1:91,1] = PR[GP1:90,1] + 34.311;
   1:  PR[GP1:91,2] = PR[GP1:90,2] + 36.483;
   1:L PR[91] R[100]mm/sec CNT100;
   1:  PR[GP1:91,1] = PR[GP1:90,1] + 30.237;
   1:  PR[GP1:91,2] = PR[GP1:90,2] + 37.985;
   1:L PR[91] R[100]mm/sec CNT100;
   1:  PR[GP1:91,1] = PR[GP1:90,1] + 19.726;
   1:  PR[GP1:91,2] = PR[GP1:90,2] + 41.433;
   1:L PR[91] R[100]mm/sec CNT100;
   1:  PR[GP1:91,1] = PR[GP1:90,1] + 16.144;
   1:  PR[GP1:91,2] = PR[GP1:90,2] + 41.498;
   1:L PR[91] R[100]mm/sec CNT100;
   1:  PR[GP1:91,1] = PR[GP1:90,1] + 4.128;
   1:  PR[GP1:91,2] = PR[GP1:90,2] + 41.067;
   1:L PR[91] R[100]mm/sec CNT100;
   1:  PR[GP1:91,1] = PR[GP1:90,1] + 1.444;
   1:  PR[GP1:91,2] = PR[GP1:90,2] + 40.247;
   1:L PR[91] R[100]mm/sec CNT100;
   1:  ! -- Layer/Ebene 154 -- !;
   1:  PR[91] = PR[90];
   1:  PR[GP1:91,1] = PR[GP1:90,1] + -1.203;
   1:  PR[GP1:91,2] = PR[GP1:90,2] + 40.421;
   1:  PR[GP1:91,3] = PR[GP1:90,3] + 94.245;
   1:L PR[91] R[100]mm/sec CNT100;
   1:  PR[GP1:91,1] = PR[GP1:90,1] + -3.615;
   1:  PR[GP1:91,2] = PR[GP1:90,2] + 41.156;
   1:L PR[91] R[100]mm/sec CNT100;
   1:  PR[GP1:91,1] = PR[GP1:90,1] + -15.968;
   1:  PR[GP1:91,2] = PR[GP1:90,2] + 41.599;
   1:L PR[91] R[100]mm/sec CNT100;
   1:  PR[GP1:91,1] = PR[GP1:90,1] + -19.250;
   1:  PR[GP1:91,2] = PR[GP1:90,2] + 41.539;
   1:L PR[91] R[100]mm/sec CNT100;
   1:  PR[GP1:91,1] = PR[GP1:90,1] + -30.091;
   1:  PR[GP1:91,2] = PR[GP1:90,2] + 37.983;
   1:L PR[91] R[100]mm/sec CNT100;
   1:  PR[GP1:91,1] = PR[GP1:90,1] + -33.876;
   1:  PR[GP1:91,2] = PR[GP1:90,2] + 36.587;
   1:L PR[91] R[100]mm/sec CNT100;
   1:  PR[GP1:91,1] = PR[GP1:90,1] + -42.097;
   1:  PR[GP1:91,2] = PR[GP1:90,2] + 30.081;
   1:L PR[91] R[100]mm/sec CNT100;
   1:  PR[GP1:91,1] = PR[GP1:90,1] + -45.706;
   1:  PR[GP1:91,2] = PR[GP1:90,2] + 27.102;
   1:L PR[91] R[100]mm/sec CNT100;
   1:  PR[GP1:91,1] = PR[GP1:90,1] + -50.732;
   1:  PR[GP1:91,2] = PR[GP1:90,2] + 18.790;
   1:L PR[91] R[100]mm/sec CNT100;
   1:  PR[GP1:91,1] = PR[GP1:90,1] + -53.360;
   1:  PR[GP1:91,2] = PR[GP1:90,2] + 14.344;
   1:L PR[91] R[100]mm/sec CNT100;
   1:  PR[GP1:91,1] = PR[GP1:90,1] + -54.342;
   1:  PR[GP1:91,2] = PR[GP1:90,2] + 8.926;
   1:L PR[91] R[100]mm/sec CNT100;
   1:  PR[GP1:91,1] = PR[GP1:90,1] + -55.530;
   1:  PR[GP1:91,2] = PR[GP1:90,2] + 1.555;
   1:L PR[91] R[100]mm/sec CNT100;
   1:  PR[GP1:91,1] = PR[GP1:90,1] + -55.831;
   1:  PR[GP1:91,2] = PR[GP1:90,2] + -0.082;
   1:L PR[91] R[100]mm/sec CNT100;
   1:  PR[GP1:91,1] = PR[GP1:90,1] + -55.028;
   1:  PR[GP1:91,2] = PR[GP1:90,2] + -5.447;
   1:L PR[91] R[100]mm/sec CNT100;
   1:  PR[GP1:91,1] = PR[GP1:90,1] + -53.360;
   1:  PR[GP1:91,2] = PR[GP1:90,2] + -14.488;
   1:L PR[91] R[100]mm/sec CNT100;
   1:  PR[GP1:91,1] = PR[GP1:90,1] + -50.731;
   1:  PR[GP1:91,2] = PR[GP1:90,2] + -18.935;
   1:L PR[91] R[100]mm/sec CNT100;
   1:  PR[GP1:91,1] = PR[GP1:90,1] + -45.705;
   1:  PR[GP1:91,2] = PR[GP1:90,2] + -27.248;
   1:L PR[91] R[100]mm/sec CNT100;
   1:  PR[GP1:91,1] = PR[GP1:90,1] + -42.094;
   1:  PR[GP1:91,2] = PR[GP1:90,2] + -30.226;
   1:L PR[91] R[100]mm/sec CNT100;
   1:  PR[GP1:91,1] = PR[GP1:90,1] + -33.874;
   1:  PR[GP1:91,2] = PR[GP1:90,2] + -36.732;
   1:L PR[91] R[100]mm/sec CNT100;
   1:  PR[GP1:91,1] = PR[GP1:90,1] + -30.089;
   1:  PR[GP1:91,2] = PR[GP1:90,2] + -38.127;
   1:L PR[91] R[100]mm/sec CNT100;
   1:  PR[GP1:91,1] = PR[GP1:90,1] + -19.248;
   1:  PR[GP1:91,2] = PR[GP1:90,2] + -41.683;
   1:L PR[91] R[100]mm/sec CNT100;
   1:  PR[GP1:91,1] = PR[GP1:90,1] + -15.966;
   1:  PR[GP1:91,2] = PR[GP1:90,2] + -41.742;
   1:L PR[91] R[100]mm/sec CNT100;
   1:  PR[GP1:91,1] = PR[GP1:90,1] + -3.619;
   1:  PR[GP1:91,2] = PR[GP1:90,2] + -41.301;
   1:L PR[91] R[100]mm/sec CNT100;
   1:  PR[GP1:91,1] = PR[GP1:90,1] + -1.205;
   1:  PR[GP1:91,2] = PR[GP1:90,2] + -40.559;
   1:L PR[91] R[100]mm/sec CNT100;
   1:  PR[GP1:91,1] = PR[GP1:90,1] + 1.420;
   1:L PR[91] R[100]mm/sec CNT100;
   1:  PR[GP1:91,1] = PR[GP1:90,1] + 3.835;
   1:  PR[GP1:91,2] = PR[GP1:90,2] + -41.301;
   1:L PR[91] R[100]mm/sec CNT100;
   1:  PR[GP1:91,1] = PR[GP1:90,1] + 16.180;
   1:  PR[GP1:91,2] = PR[GP1:90,2] + -41.741;
   1:L PR[91] R[100]mm/sec CNT100;
   1:  PR[GP1:91,1] = PR[GP1:90,1] + 19.463;
   1:  PR[GP1:91,2] = PR[GP1:90,2] + -41.683;
   1:L PR[91] R[100]mm/sec CNT100;
   1:  PR[GP1:91,1] = PR[GP1:90,1] + 30.302;
   1:  PR[GP1:91,2] = PR[GP1:90,2] + -38.127;
   1:L PR[91] R[100]mm/sec CNT100;
   1:  PR[GP1:91,1] = PR[GP1:90,1] + 34.088;
   1:  PR[GP1:91,2] = PR[GP1:90,2] + -36.733;
   1:L PR[91] R[100]mm/sec CNT100;
   1:  PR[GP1:91,1] = PR[GP1:90,1] + 42.307;
   1:  PR[GP1:91,2] = PR[GP1:90,2] + -30.226;
   1:L PR[91] R[100]mm/sec CNT100;
   1:  PR[GP1:91,1] = PR[GP1:90,1] + 45.918;
   1:  PR[GP1:91,2] = PR[GP1:90,2] + -27.244;
   1:L PR[91] R[100]mm/sec CNT100;
   1:  PR[GP1:91,1] = PR[GP1:90,1] + 50.944;
   1:  PR[GP1:91,2] = PR[GP1:90,2] + -18.935;
   1:L PR[91] R[100]mm/sec CNT100;
   1:  PR[GP1:91,1] = PR[GP1:90,1] + 53.572;
   1:  PR[GP1:91,2] = PR[GP1:90,2] + -14.499;
   1:L PR[91] R[100]mm/sec CNT100;
   1:  PR[GP1:91,1] = PR[GP1:90,1] + 54.555;
   1:  PR[GP1:91,2] = PR[GP1:90,2] + -9.073;
   1:L PR[91] R[100]mm/sec CNT100;
   1:  PR[GP1:91,1] = PR[GP1:90,1] + 55.743;
   1:  PR[GP1:91,2] = PR[GP1:90,2] + -1.700;
   1:L PR[91] R[100]mm/sec CNT100;
   1:  PR[GP1:91,1] = PR[GP1:90,1] + 56.044;
   1:  PR[GP1:91,2] = PR[GP1:90,2] + -0.062;
   1:L PR[91] R[100]mm/sec CNT100;
   1:  PR[GP1:91,1] = PR[GP1:90,1] + 55.241;
   1:  PR[GP1:91,2] = PR[GP1:90,2] + 5.309;
   1:L PR[91] R[100]mm/sec CNT100;
   1:  PR[GP1:91,1] = PR[GP1:90,1] + 53.573;
   1:  PR[GP1:91,2] = PR[GP1:90,2] + 14.353;
   1:L PR[91] R[100]mm/sec CNT100;
   1:  PR[GP1:91,1] = PR[GP1:90,1] + 50.946;
   1:  PR[GP1:91,2] = PR[GP1:90,2] + 18.790;
   1:L PR[91] R[100]mm/sec CNT100;
   1:  PR[GP1:91,1] = PR[GP1:90,1] + 45.920;
   1:  PR[GP1:91,2] = PR[GP1:90,2] + 27.098;
   1:L PR[91] R[100]mm/sec CNT100;
   1:  PR[GP1:91,1] = PR[GP1:90,1] + 42.310;
   1:  PR[GP1:91,2] = PR[GP1:90,2] + 30.081;
   1:L PR[91] R[100]mm/sec CNT100;
   1:  PR[GP1:91,1] = PR[GP1:90,1] + 34.090;
   1:  PR[GP1:91,2] = PR[GP1:90,2] + 36.588;
   1:L PR[91] R[100]mm/sec CNT100;
   1:  PR[GP1:91,1] = PR[GP1:90,1] + 30.305;
   1:  PR[GP1:91,2] = PR[GP1:90,2] + 37.983;
   1:L PR[91] R[100]mm/sec CNT100;
   1:  PR[GP1:91,1] = PR[GP1:90,1] + 19.464;
   1:  PR[GP1:91,2] = PR[GP1:90,2] + 41.539;
   1:L PR[91] R[100]mm/sec CNT100;
   1:  PR[GP1:91,1] = PR[GP1:90,1] + 16.182;
   1:  PR[GP1:91,2] = PR[GP1:90,2] + 41.598;
   1:L PR[91] R[100]mm/sec CNT100;
   1:  PR[GP1:91,1] = PR[GP1:90,1] + 3.831;
   1:  PR[GP1:91,2] = PR[GP1:90,2] + 41.156;
   1:L PR[91] R[100]mm/sec CNT100;
   1:  PR[GP1:91,1] = PR[GP1:90,1] + 1.418;
   1:  PR[GP1:91,2] = PR[GP1:90,2] + 40.420;
   1:L PR[91] R[100]mm/sec CNT100;
   1:  ! -- Layer/Ebene 155 -- !;
   1:  PR[91] = PR[90];
   1:  PR[GP1:91,1] = PR[GP1:90,1] + -1.178;
   1:  PR[GP1:91,2] = PR[GP1:90,2] + 40.594;
   1:  PR[GP1:91,3] = PR[GP1:90,3] + 94.855;
   1:L PR[91] R[100]mm/sec CNT100;
   1:  PR[GP1:91,1] = PR[GP1:90,1] + -3.318;
   1:  PR[GP1:91,2] = PR[GP1:90,2] + 41.244;
   1:L PR[91] R[100]mm/sec CNT100;
   1:  PR[GP1:91,1] = PR[GP1:90,1] + -16.006;
   1:  PR[GP1:91,2] = PR[GP1:90,2] + 41.700;
   1:L PR[91] R[100]mm/sec CNT100;
   1:  PR[GP1:91,1] = PR[GP1:90,1] + -18.988;
   1:  PR[GP1:91,2] = PR[GP1:90,2] + 41.645;
   1:L PR[91] R[100]mm/sec CNT100;
   1:  PR[GP1:91,1] = PR[GP1:90,1] + -30.160;
   1:  PR[GP1:91,2] = PR[GP1:90,2] + 37.981;
   1:L PR[91] R[100]mm/sec CNT100;
   1:  PR[GP1:91,1] = PR[GP1:90,1] + -33.654;
   1:  PR[GP1:91,2] = PR[GP1:90,2] + 36.692;
   1:L PR[91] R[100]mm/sec CNT100;
   1:  PR[GP1:91,1] = PR[GP1:90,1] + -42.157;
   1:  PR[GP1:91,2] = PR[GP1:90,2] + 29.964;
   1:L PR[91] R[100]mm/sec CNT100;
   1:  PR[GP1:91,1] = PR[GP1:90,1] + -45.522;
   1:  PR[GP1:91,2] = PR[GP1:90,2] + 27.187;
   1:L PR[91] R[100]mm/sec CNT100;
   1:  PR[GP1:91,1] = PR[GP1:90,1] + -50.739;
   1:  PR[GP1:91,2] = PR[GP1:90,2] + 18.557;
   1:L PR[91] R[100]mm/sec CNT100;
   1:  PR[GP1:91,1] = PR[GP1:90,1] + -53.201;
   1:  PR[GP1:91,2] = PR[GP1:90,2] + 14.391;
   1:L PR[91] R[100]mm/sec CNT100;
   1:  PR[GP1:91,1] = PR[GP1:90,1] + -54.121;
   1:  PR[GP1:91,2] = PR[GP1:90,2] + 9.314;
   1:L PR[91] R[100]mm/sec CNT100;
   1:  PR[GP1:91,1] = PR[GP1:90,1] + -55.236;
   1:  PR[GP1:91,2] = PR[GP1:90,2] + 2.398;
   1:L PR[91] R[100]mm/sec CNT100;
   1:  PR[GP1:91,1] = PR[GP1:90,1] + -55.693;
   1:  PR[GP1:91,2] = PR[GP1:90,2] + -0.082;
   1:L PR[91] R[100]mm/sec CNT100;
   1:  PR[GP1:91,1] = PR[GP1:90,1] + -54.938;
   1:  PR[GP1:91,2] = PR[GP1:90,2] + -5.122;
   1:L PR[91] R[100]mm/sec CNT100;
   1:  PR[GP1:91,1] = PR[GP1:90,1] + -53.201;
   1:  PR[GP1:91,2] = PR[GP1:90,2] + -14.535;
   1:L PR[91] R[100]mm/sec CNT100;
   1:  PR[GP1:91,1] = PR[GP1:90,1] + -50.738;
   1:  PR[GP1:91,2] = PR[GP1:90,2] + -18.702;
   1:L PR[91] R[100]mm/sec CNT100;
   1:  PR[GP1:91,1] = PR[GP1:90,1] + -45.520;
   1:  PR[GP1:91,2] = PR[GP1:90,2] + -27.332;
   1:L PR[91] R[100]mm/sec CNT100;
   1:  PR[GP1:91,1] = PR[GP1:90,1] + -42.154;
   1:  PR[GP1:91,2] = PR[GP1:90,2] + -30.109;
   1:L PR[91] R[100]mm/sec CNT100;
   1:  PR[GP1:91,1] = PR[GP1:90,1] + -33.653;
   1:  PR[GP1:91,2] = PR[GP1:90,2] + -36.837;
   1:L PR[91] R[100]mm/sec CNT100;
   1:  PR[GP1:91,1] = PR[GP1:90,1] + -30.158;
   1:  PR[GP1:91,2] = PR[GP1:90,2] + -38.125;
   1:L PR[91] R[100]mm/sec CNT100;
   1:  PR[GP1:91,1] = PR[GP1:90,1] + -18.988;
   1:  PR[GP1:91,2] = PR[GP1:90,2] + -41.789;
   1:L PR[91] R[100]mm/sec CNT100;
   1:  PR[GP1:91,1] = PR[GP1:90,1] + -16.005;
   1:  PR[GP1:91,2] = PR[GP1:90,2] + -41.842;
   1:L PR[91] R[100]mm/sec CNT100;
   1:  PR[GP1:91,1] = PR[GP1:90,1] + -3.322;
   1:  PR[GP1:91,2] = PR[GP1:90,2] + -41.390;
   1:L PR[91] R[100]mm/sec CNT100;
   1:  PR[GP1:91,1] = PR[GP1:90,1] + -1.179;
   1:  PR[GP1:91,2] = PR[GP1:90,2] + -40.733;
   1:L PR[91] R[100]mm/sec CNT100;
   1:  PR[GP1:91,1] = PR[GP1:90,1] + 1.394;
   1:L PR[91] R[100]mm/sec CNT100;
   1:  PR[GP1:91,1] = PR[GP1:90,1] + 3.538;
   1:  PR[GP1:91,2] = PR[GP1:90,2] + -41.390;
   1:L PR[91] R[100]mm/sec CNT100;
   1:  PR[GP1:91,1] = PR[GP1:90,1] + 16.219;
   1:  PR[GP1:91,2] = PR[GP1:90,2] + -41.842;
   1:L PR[91] R[100]mm/sec CNT100;
   1:  PR[GP1:91,1] = PR[GP1:90,1] + 19.202;
   1:  PR[GP1:91,2] = PR[GP1:90,2] + -41.789;
   1:L PR[91] R[100]mm/sec CNT100;
   1:  PR[GP1:91,1] = PR[GP1:90,1] + 30.371;
   1:  PR[GP1:91,2] = PR[GP1:90,2] + -38.125;
   1:L PR[91] R[100]mm/sec CNT100;
   1:  PR[GP1:91,1] = PR[GP1:90,1] + 33.867;
   1:  PR[GP1:91,2] = PR[GP1:90,2] + -36.837;
   1:L PR[91] R[100]mm/sec CNT100;
   1:  PR[GP1:91,1] = PR[GP1:90,1] + 42.368;
   1:  PR[GP1:91,2] = PR[GP1:90,2] + -30.107;
   1:L PR[91] R[100]mm/sec CNT100;
   1:  PR[GP1:91,1] = PR[GP1:90,1] + 45.734;
   1:  PR[GP1:91,2] = PR[GP1:90,2] + -27.328;
   1:L PR[91] R[100]mm/sec CNT100;
   1:  PR[GP1:91,1] = PR[GP1:90,1] + 50.951;
   1:  PR[GP1:91,2] = PR[GP1:90,2] + -18.703;
   1:L PR[91] R[100]mm/sec CNT100;
   1:  PR[GP1:91,1] = PR[GP1:90,1] + 53.414;
   1:  PR[GP1:91,2] = PR[GP1:90,2] + -14.546;
   1:L PR[91] R[100]mm/sec CNT100;
   1:  PR[GP1:91,1] = PR[GP1:90,1] + 54.335;
   1:  PR[GP1:91,2] = PR[GP1:90,2] + -9.461;
   1:L PR[91] R[100]mm/sec CNT100;
   1:  PR[GP1:91,1] = PR[GP1:90,1] + 55.450;
   1:  PR[GP1:91,2] = PR[GP1:90,2] + -2.542;
   1:L PR[91] R[100]mm/sec CNT100;
   1:  PR[GP1:91,1] = PR[GP1:90,1] + 55.906;
   1:  PR[GP1:91,2] = PR[GP1:90,2] + -0.062;
   1:L PR[91] R[100]mm/sec CNT100;
   1:  PR[GP1:91,1] = PR[GP1:90,1] + 55.152;
   1:  PR[GP1:91,2] = PR[GP1:90,2] + 4.983;
   1:L PR[91] R[100]mm/sec CNT100;
   1:  PR[GP1:91,1] = PR[GP1:90,1] + 53.415;
   1:  PR[GP1:91,2] = PR[GP1:90,2] + 14.400;
   1:L PR[91] R[100]mm/sec CNT100;
   1:  PR[GP1:91,1] = PR[GP1:90,1] + 50.953;
   1:  PR[GP1:91,2] = PR[GP1:90,2] + 18.557;
   1:L PR[91] R[100]mm/sec CNT100;
   1:  PR[GP1:91,1] = PR[GP1:90,1] + 45.735;
   1:  PR[GP1:91,2] = PR[GP1:90,2] + 27.183;
   1:L PR[91] R[100]mm/sec CNT100;
   1:  PR[GP1:91,1] = PR[GP1:90,1] + 42.370;
   1:  PR[GP1:91,2] = PR[GP1:90,2] + 29.963;
   1:L PR[91] R[100]mm/sec CNT100;
   1:  PR[GP1:91,1] = PR[GP1:90,1] + 33.868;
   1:  PR[GP1:91,2] = PR[GP1:90,2] + 36.693;
   1:L PR[91] R[100]mm/sec CNT100;
   1:  PR[GP1:91,1] = PR[GP1:90,1] + 30.374;
   1:  PR[GP1:91,2] = PR[GP1:90,2] + 37.981;
   1:L PR[91] R[100]mm/sec CNT100;
   1:  PR[GP1:91,1] = PR[GP1:90,1] + 19.203;
   1:  PR[GP1:91,2] = PR[GP1:90,2] + 41.645;
   1:L PR[91] R[100]mm/sec CNT100;
   1:  PR[GP1:91,1] = PR[GP1:90,1] + 16.221;
   1:  PR[GP1:91,2] = PR[GP1:90,2] + 41.699;
   1:L PR[91] R[100]mm/sec CNT100;
   1:  PR[GP1:91,1] = PR[GP1:90,1] + 3.533;
   1:  PR[GP1:91,2] = PR[GP1:90,2] + 41.244;
   1:L PR[91] R[100]mm/sec CNT100;
   1:  PR[GP1:91,1] = PR[GP1:90,1] + 1.393;
   1:  PR[GP1:91,2] = PR[GP1:90,2] + 40.594;
   1:L PR[91] R[100]mm/sec CNT100;
   1:  ! -- Layer/Ebene 156 -- !;
   1:  PR[91] = PR[90];
   1:  PR[GP1:91,1] = PR[GP1:90,1] + -1.152;
   1:  PR[GP1:91,2] = PR[GP1:90,2] + 40.767;
   1:  PR[GP1:91,3] = PR[GP1:90,3] + 95.465;
   1:L PR[91] R[100]mm/sec CNT100;
   1:  PR[GP1:91,1] = PR[GP1:90,1] + -3.020;
   1:  PR[GP1:91,2] = PR[GP1:90,2] + 41.333;
   1:L PR[91] R[100]mm/sec CNT100;
   1:  PR[GP1:91,1] = PR[GP1:90,1] + -16.044;
   1:  PR[GP1:91,2] = PR[GP1:90,2] + 41.800;
   1:L PR[91] R[100]mm/sec CNT100;
   1:  PR[GP1:91,1] = PR[GP1:90,1] + -18.727;
   1:  PR[GP1:91,2] = PR[GP1:90,2] + 41.751;
   1:L PR[91] R[100]mm/sec CNT100;
   1:  PR[GP1:91,1] = PR[GP1:90,1] + -30.228;
   1:  PR[GP1:91,2] = PR[GP1:90,2] + 37.979;
   1:L PR[91] R[100]mm/sec CNT100;
   1:  PR[GP1:91,1] = PR[GP1:90,1] + -33.433;
   1:  PR[GP1:91,2] = PR[GP1:90,2] + 36.797;
   1:L PR[91] R[100]mm/sec CNT100;
   1:  PR[GP1:91,1] = PR[GP1:90,1] + -42.217;
   1:  PR[GP1:91,2] = PR[GP1:90,2] + 29.846;
   1:L PR[91] R[100]mm/sec CNT100;
   1:  PR[GP1:91,1] = PR[GP1:90,1] + -45.337;
   1:  PR[GP1:91,2] = PR[GP1:90,2] + 27.271;
   1:L PR[91] R[100]mm/sec CNT100;
   1:  PR[GP1:91,1] = PR[GP1:90,1] + -50.747;
   1:  PR[GP1:91,2] = PR[GP1:90,2] + 18.324;
   1:L PR[91] R[100]mm/sec CNT100;
   1:  PR[GP1:91,1] = PR[GP1:90,1] + -53.042;
   1:  PR[GP1:91,2] = PR[GP1:90,2] + 14.438;
   1:L PR[91] R[100]mm/sec CNT100;
   1:  PR[GP1:91,1] = PR[GP1:90,1] + -53.901;
   1:  PR[GP1:91,2] = PR[GP1:90,2] + 9.702;
   1:L PR[91] R[100]mm/sec CNT100;
   1:  PR[GP1:91,1] = PR[GP1:90,1] + -54.943;
   1:  PR[GP1:91,2] = PR[GP1:90,2] + 3.240;
   1:L PR[91] R[100]mm/sec CNT100;
   1:  PR[GP1:91,1] = PR[GP1:90,1] + -55.554;
   1:  PR[GP1:91,2] = PR[GP1:90,2] + -0.082;
   1:L PR[91] R[100]mm/sec CNT100;
   1:  PR[GP1:91,1] = PR[GP1:90,1] + -54.848;
   1:  PR[GP1:91,2] = PR[GP1:90,2] + -4.796;
   1:L PR[91] R[100]mm/sec CNT100;
   1:  PR[GP1:91,1] = PR[GP1:90,1] + -53.043;
   1:  PR[GP1:91,2] = PR[GP1:90,2] + -14.582;
   1:L PR[91] R[100]mm/sec CNT100;
   1:  PR[GP1:91,1] = PR[GP1:90,1] + -50.745;
   1:  PR[GP1:91,2] = PR[GP1:90,2] + -18.469;
   1:L PR[91] R[100]mm/sec CNT100;
   1:  PR[GP1:91,1] = PR[GP1:90,1] + -45.336;
   1:  PR[GP1:91,2] = PR[GP1:90,2] + -27.416;
   1:L PR[91] R[100]mm/sec CNT100;
   1:  PR[GP1:91,1] = PR[GP1:90,1] + -42.214;
   1:  PR[GP1:91,2] = PR[GP1:90,2] + -29.991;
   1:L PR[91] R[100]mm/sec CNT100;
   1:  PR[GP1:91,1] = PR[GP1:90,1] + -33.432;
   1:  PR[GP1:91,2] = PR[GP1:90,2] + -36.941;
   1:L PR[91] R[100]mm/sec CNT100;
   1:  PR[GP1:91,1] = PR[GP1:90,1] + -30.227;
   1:  PR[GP1:91,2] = PR[GP1:90,2] + -38.123;
   1:L PR[91] R[100]mm/sec CNT100;
   1:  PR[GP1:91,1] = PR[GP1:90,1] + -18.727;
   1:  PR[GP1:91,2] = PR[GP1:90,2] + -41.895;
   1:L PR[91] R[100]mm/sec CNT100;
   1:  PR[GP1:91,1] = PR[GP1:90,1] + -16.043;
   1:  PR[GP1:91,2] = PR[GP1:90,2] + -41.943;
   1:L PR[91] R[100]mm/sec CNT100;
   1:  PR[GP1:91,1] = PR[GP1:90,1] + -3.025;
   1:  PR[GP1:91,2] = PR[GP1:90,2] + -41.479;
   1:L PR[91] R[100]mm/sec CNT100;
   1:  PR[GP1:91,1] = PR[GP1:90,1] + -1.154;
   1:  PR[GP1:91,2] = PR[GP1:90,2] + -40.906;
   1:L PR[91] R[100]mm/sec CNT100;
   1:  PR[GP1:91,1] = PR[GP1:90,1] + 1.369;
   1:L PR[91] R[100]mm/sec CNT100;
   1:  PR[GP1:91,1] = PR[GP1:90,1] + 3.241;
   1:  PR[GP1:91,2] = PR[GP1:90,2] + -41.479;
   1:L PR[91] R[100]mm/sec CNT100;
   1:  PR[GP1:91,1] = PR[GP1:90,1] + 16.258;
   1:  PR[GP1:91,2] = PR[GP1:90,2] + -41.943;
   1:L PR[91] R[100]mm/sec CNT100;
   1:  PR[GP1:91,1] = PR[GP1:90,1] + 18.942;
   1:  PR[GP1:91,2] = PR[GP1:90,2] + -41.895;
   1:L PR[91] R[100]mm/sec CNT100;
   1:  PR[GP1:91,1] = PR[GP1:90,1] + 30.440;
   1:  PR[GP1:91,2] = PR[GP1:90,2] + -38.123;
   1:L PR[91] R[100]mm/sec CNT100;
   1:  PR[GP1:91,1] = PR[GP1:90,1] + 33.646;
   1:  PR[GP1:91,2] = PR[GP1:90,2] + -36.942;
   1:L PR[91] R[100]mm/sec CNT100;
   1:  PR[GP1:91,1] = PR[GP1:90,1] + 42.428;
   1:  PR[GP1:91,2] = PR[GP1:90,2] + -29.989;
   1:L PR[91] R[100]mm/sec CNT100;
   1:  PR[GP1:91,1] = PR[GP1:90,1] + 45.550;
   1:  PR[GP1:91,2] = PR[GP1:90,2] + -27.412;
   1:L PR[91] R[100]mm/sec CNT100;
   1:  PR[GP1:91,1] = PR[GP1:90,1] + 50.958;
   1:  PR[GP1:91,2] = PR[GP1:90,2] + -18.470;
   1:L PR[91] R[100]mm/sec CNT100;
   1:  PR[GP1:91,1] = PR[GP1:90,1] + 53.256;
   1:  PR[GP1:91,2] = PR[GP1:90,2] + -14.592;
   1:L PR[91] R[100]mm/sec CNT100;
   1:  PR[GP1:91,1] = PR[GP1:90,1] + 54.115;
   1:  PR[GP1:91,2] = PR[GP1:90,2] + -9.849;
   1:L PR[91] R[100]mm/sec CNT100;
   1:  PR[GP1:91,1] = PR[GP1:90,1] + 55.156;
   1:  PR[GP1:91,2] = PR[GP1:90,2] + -3.385;
   1:L PR[91] R[100]mm/sec CNT100;
   1:  PR[GP1:91,1] = PR[GP1:90,1] + 55.768;
   1:  PR[GP1:91,2] = PR[GP1:90,2] + -0.062;
   1:L PR[91] R[100]mm/sec CNT100;
   1:  PR[GP1:91,1] = PR[GP1:90,1] + 55.062;
   1:  PR[GP1:91,2] = PR[GP1:90,2] + 4.657;
   1:L PR[91] R[100]mm/sec CNT100;
   1:  PR[GP1:91,1] = PR[GP1:90,1] + 53.256;
   1:  PR[GP1:91,2] = PR[GP1:90,2] + 14.447;
   1:L PR[91] R[100]mm/sec CNT100;
   1:  PR[GP1:91,1] = PR[GP1:90,1] + 50.960;
   1:  PR[GP1:91,2] = PR[GP1:90,2] + 18.325;
   1:L PR[91] R[100]mm/sec CNT100;
   1:  PR[GP1:91,1] = PR[GP1:90,1] + 45.550;
   1:  PR[GP1:91,2] = PR[GP1:90,2] + 27.267;
   1:L PR[91] R[100]mm/sec CNT100;
   1:  PR[GP1:91,1] = PR[GP1:90,1] + 42.430;
   1:  PR[GP1:91,2] = PR[GP1:90,2] + 29.845;
   1:L PR[91] R[100]mm/sec CNT100;
   1:  PR[GP1:91,1] = PR[GP1:90,1] + 33.647;
   1:  PR[GP1:91,2] = PR[GP1:90,2] + 36.797;
   1:L PR[91] R[100]mm/sec CNT100;
   1:  PR[GP1:91,1] = PR[GP1:90,1] + 30.442;
   1:  PR[GP1:91,2] = PR[GP1:90,2] + 37.979;
   1:L PR[91] R[100]mm/sec CNT100;
   1:  PR[GP1:91,1] = PR[GP1:90,1] + 18.942;
   1:  PR[GP1:91,2] = PR[GP1:90,2] + 41.751;
   1:L PR[91] R[100]mm/sec CNT100;
   1:  PR[GP1:91,1] = PR[GP1:90,1] + 16.259;
   1:  PR[GP1:91,2] = PR[GP1:90,2] + 41.800;
   1:L PR[91] R[100]mm/sec CNT100;
   1:  PR[GP1:91,1] = PR[GP1:90,1] + 3.235;
   1:  PR[GP1:91,2] = PR[GP1:90,2] + 41.333;
   1:L PR[91] R[100]mm/sec CNT100;
   1:  PR[GP1:91,1] = PR[GP1:90,1] + 1.368;
   1:  PR[GP1:91,2] = PR[GP1:90,2] + 40.767;
   1:L PR[91] R[100]mm/sec CNT100;
   1:  ! -- Layer/Ebene 157 -- !;
   1:  PR[91] = PR[90];
   1:  PR[GP1:91,1] = PR[GP1:90,1] + -1.126;
   1:  PR[GP1:91,2] = PR[GP1:90,2] + 40.940;
   1:  PR[GP1:91,3] = PR[GP1:90,3] + 96.075;
   1:L PR[91] R[100]mm/sec CNT100;
   1:  PR[GP1:91,1] = PR[GP1:90,1] + -2.722;
   1:  PR[GP1:91,2] = PR[GP1:90,2] + 41.422;
   1:L PR[91] R[100]mm/sec CNT100;
   1:  PR[GP1:91,1] = PR[GP1:90,1] + -16.082;
   1:  PR[GP1:91,2] = PR[GP1:90,2] + 41.901;
   1:L PR[91] R[100]mm/sec CNT100;
   1:  PR[GP1:91,1] = PR[GP1:90,1] + -18.466;
   1:  PR[GP1:91,2] = PR[GP1:90,2] + 41.857;
   1:L PR[91] R[100]mm/sec CNT100;
   1:  PR[GP1:91,1] = PR[GP1:90,1] + -30.297;
   1:  PR[GP1:91,2] = PR[GP1:90,2] + 37.977;
   1:L PR[91] R[100]mm/sec CNT100;
   1:  PR[GP1:91,1] = PR[GP1:90,1] + -33.211;
   1:  PR[GP1:91,2] = PR[GP1:90,2] + 36.902;
   1:L PR[91] R[100]mm/sec CNT100;
   1:  PR[GP1:91,1] = PR[GP1:90,1] + -42.277;
   1:  PR[GP1:91,2] = PR[GP1:90,2] + 29.728;
   1:L PR[91] R[100]mm/sec CNT100;
   1:  PR[GP1:91,1] = PR[GP1:90,1] + -45.152;
   1:  PR[GP1:91,2] = PR[GP1:90,2] + 27.355;
   1:L PR[91] R[100]mm/sec CNT100;
   1:  PR[GP1:91,1] = PR[GP1:90,1] + -50.753;
   1:  PR[GP1:91,2] = PR[GP1:90,2] + 18.091;
   1:L PR[91] R[100]mm/sec CNT100;
   1:  PR[GP1:91,1] = PR[GP1:90,1] + -52.884;
   1:  PR[GP1:91,2] = PR[GP1:90,2] + 14.486;
   1:L PR[91] R[100]mm/sec CNT100;
   1:  PR[GP1:91,1] = PR[GP1:90,1] + -53.681;
   1:  PR[GP1:91,2] = PR[GP1:90,2] + 10.091;
   1:L PR[91] R[100]mm/sec CNT100;
   1:  PR[GP1:91,1] = PR[GP1:90,1] + -54.649;
   1:  PR[GP1:91,2] = PR[GP1:90,2] + 4.083;
   1:L PR[91] R[100]mm/sec CNT100;
   1:  PR[GP1:91,1] = PR[GP1:90,1] + -55.416;
   1:  PR[GP1:91,2] = PR[GP1:90,2] + -0.082;
   1:L PR[91] R[100]mm/sec CNT100;
   1:  PR[GP1:91,1] = PR[GP1:90,1] + -54.759;
   1:  PR[GP1:91,2] = PR[GP1:90,2] + -4.470;
   1:L PR[91] R[100]mm/sec CNT100;
   1:  PR[GP1:91,1] = PR[GP1:90,1] + -52.884;
   1:  PR[GP1:91,2] = PR[GP1:90,2] + -14.629;
   1:L PR[91] R[100]mm/sec CNT100;
   1:  PR[GP1:91,1] = PR[GP1:90,1] + -50.752;
   1:  PR[GP1:91,2] = PR[GP1:90,2] + -18.237;
   1:L PR[91] R[100]mm/sec CNT100;
   1:  PR[GP1:91,1] = PR[GP1:90,1] + -45.151;
   1:  PR[GP1:91,2] = PR[GP1:90,2] + -27.500;
   1:L PR[91] R[100]mm/sec CNT100;
   1:  PR[GP1:91,1] = PR[GP1:90,1] + -42.274;
   1:  PR[GP1:91,2] = PR[GP1:90,2] + -29.873;
   1:L PR[91] R[100]mm/sec CNT100;
   1:  PR[GP1:91,1] = PR[GP1:90,1] + -33.210;
   1:  PR[GP1:91,2] = PR[GP1:90,2] + -37.046;
   1:L PR[91] R[100]mm/sec CNT100;
   1:  PR[GP1:91,1] = PR[GP1:90,1] + -30.295;
   1:  PR[GP1:91,2] = PR[GP1:90,2] + -38.121;
   1:L PR[91] R[100]mm/sec CNT100;
   1:  PR[GP1:91,1] = PR[GP1:90,1] + -18.466;
   1:  PR[GP1:91,2] = PR[GP1:90,2] + -42.001;
   1:L PR[91] R[100]mm/sec CNT100;
   1:  PR[GP1:91,1] = PR[GP1:90,1] + -16.082;
   1:  PR[GP1:91,2] = PR[GP1:90,2] + -42.044;
   1:L PR[91] R[100]mm/sec CNT100;
   1:  PR[GP1:91,1] = PR[GP1:90,1] + -2.728;
   1:  PR[GP1:91,2] = PR[GP1:90,2] + -41.568;
   1:L PR[91] R[100]mm/sec CNT100;
   1:  PR[GP1:91,1] = PR[GP1:90,1] + -1.128;
   1:  PR[GP1:91,2] = PR[GP1:90,2] + -41.080;
   1:L PR[91] R[100]mm/sec CNT100;
   1:  PR[GP1:91,1] = PR[GP1:90,1] + 1.344;
   1:L PR[91] R[100]mm/sec CNT100;
   1:  PR[GP1:91,1] = PR[GP1:90,1] + 2.944;
   1:  PR[GP1:91,2] = PR[GP1:90,2] + -41.568;
   1:L PR[91] R[100]mm/sec CNT100;
   1:  PR[GP1:91,1] = PR[GP1:90,1] + 16.297;
   1:  PR[GP1:91,2] = PR[GP1:90,2] + -42.043;
   1:L PR[91] R[100]mm/sec CNT100;
   1:  PR[GP1:91,1] = PR[GP1:90,1] + 18.681;
   1:  PR[GP1:91,2] = PR[GP1:90,2] + -42.001;
   1:L PR[91] R[100]mm/sec CNT100;
   1:  PR[GP1:91,1] = PR[GP1:90,1] + 30.509;
   1:  PR[GP1:91,2] = PR[GP1:90,2] + -38.121;
   1:L PR[91] R[100]mm/sec CNT100;
   1:  PR[GP1:91,1] = PR[GP1:90,1] + 33.425;
   1:  PR[GP1:91,2] = PR[GP1:90,2] + -37.047;
   1:L PR[91] R[100]mm/sec CNT100;
   1:  PR[GP1:91,1] = PR[GP1:90,1] + 42.488;
   1:  PR[GP1:91,2] = PR[GP1:90,2] + -29.872;
   1:L PR[91] R[100]mm/sec CNT100;
   1:  PR[GP1:91,1] = PR[GP1:90,1] + 45.365;
   1:  PR[GP1:91,2] = PR[GP1:90,2] + -27.496;
   1:L PR[91] R[100]mm/sec CNT100;
   1:  PR[GP1:91,1] = PR[GP1:90,1] + 50.965;
   1:  PR[GP1:91,2] = PR[GP1:90,2] + -18.237;
   1:L PR[91] R[100]mm/sec CNT100;
   1:  PR[GP1:91,1] = PR[GP1:90,1] + 53.097;
   1:  PR[GP1:91,2] = PR[GP1:90,2] + -14.639;
   1:L PR[91] R[100]mm/sec CNT100;
   1:  PR[GP1:91,1] = PR[GP1:90,1] + 53.894;
   1:  PR[GP1:91,2] = PR[GP1:90,2] + -10.237;
   1:L PR[91] R[100]mm/sec CNT100;
   1:  PR[GP1:91,1] = PR[GP1:90,1] + 54.863;
   1:  PR[GP1:91,2] = PR[GP1:90,2] + -4.228;
   1:L PR[91] R[100]mm/sec CNT100;
   1:  PR[GP1:91,1] = PR[GP1:90,1] + 55.629;
   1:  PR[GP1:91,2] = PR[GP1:90,2] + -0.062;
   1:L PR[91] R[100]mm/sec CNT100;
   1:  PR[GP1:91,1] = PR[GP1:90,1] + 54.972;
   1:  PR[GP1:91,2] = PR[GP1:90,2] + 4.332;
   1:L PR[91] R[100]mm/sec CNT100;
   1:  PR[GP1:91,1] = PR[GP1:90,1] + 53.098;
   1:  PR[GP1:91,2] = PR[GP1:90,2] + 14.494;
   1:L PR[91] R[100]mm/sec CNT100;
   1:  PR[GP1:91,1] = PR[GP1:90,1] + 50.967;
   1:  PR[GP1:91,2] = PR[GP1:90,2] + 18.092;
   1:L PR[91] R[100]mm/sec CNT100;
   1:  PR[GP1:91,1] = PR[GP1:90,1] + 45.366;
   1:  PR[GP1:91,2] = PR[GP1:90,2] + 27.351;
   1:L PR[91] R[100]mm/sec CNT100;
   1:  PR[GP1:91,1] = PR[GP1:90,1] + 42.490;
   1:  PR[GP1:91,2] = PR[GP1:90,2] + 29.727;
   1:L PR[91] R[100]mm/sec CNT100;
   1:  PR[GP1:91,1] = PR[GP1:90,1] + 33.425;
   1:  PR[GP1:91,2] = PR[GP1:90,2] + 36.902;
   1:L PR[91] R[100]mm/sec CNT100;
   1:  PR[GP1:91,1] = PR[GP1:90,1] + 30.511;
   1:  PR[GP1:91,2] = PR[GP1:90,2] + 37.977;
   1:L PR[91] R[100]mm/sec CNT100;
   1:  PR[GP1:91,1] = PR[GP1:90,1] + 18.681;
   1:  PR[GP1:91,2] = PR[GP1:90,2] + 41.857;
   1:L PR[91] R[100]mm/sec CNT100;
   1:  PR[GP1:91,1] = PR[GP1:90,1] + 16.297;
   1:  PR[GP1:91,2] = PR[GP1:90,2] + 41.901;
   1:L PR[91] R[100]mm/sec CNT100;
   1:  PR[GP1:91,1] = PR[GP1:90,1] + 2.937;
   1:  PR[GP1:91,2] = PR[GP1:90,2] + 41.422;
   1:L PR[91] R[100]mm/sec CNT100;
   1:  PR[GP1:91,1] = PR[GP1:90,1] + 1.342;
   1:  PR[GP1:91,2] = PR[GP1:90,2] + 40.940;
   1:L PR[91] R[100]mm/sec CNT100;
   1:  ! -- Layer/Ebene 158 -- !;
   1:  PR[91] = PR[90];
   1:  PR[GP1:91,1] = PR[GP1:90,1] + -1.101;
   1:  PR[GP1:91,2] = PR[GP1:90,2] + 41.113;
   1:  PR[GP1:91,3] = PR[GP1:90,3] + 96.685;
   1:L PR[91] R[100]mm/sec CNT100;
   1:  PR[GP1:91,1] = PR[GP1:90,1] + -2.424;
   1:  PR[GP1:91,2] = PR[GP1:90,2] + 41.510;
   1:L PR[91] R[100]mm/sec CNT100;
   1:  PR[GP1:91,1] = PR[GP1:90,1] + -16.120;
   1:  PR[GP1:91,2] = PR[GP1:90,2] + 42.002;
   1:L PR[91] R[100]mm/sec CNT100;
   1:  PR[GP1:91,1] = PR[GP1:90,1] + -18.204;
   1:  PR[GP1:91,2] = PR[GP1:90,2] + 41.964;
   1:L PR[91] R[100]mm/sec CNT100;
   1:  PR[GP1:91,1] = PR[GP1:90,1] + -30.365;
   1:  PR[GP1:91,2] = PR[GP1:90,2] + 37.975;
   1:L PR[91] R[100]mm/sec CNT100;
   1:  PR[GP1:91,1] = PR[GP1:90,1] + -32.990;
   1:  PR[GP1:91,2] = PR[GP1:90,2] + 37.007;
   1:L PR[91] R[100]mm/sec CNT100;
   1:  PR[GP1:91,1] = PR[GP1:90,1] + -42.336;
   1:  PR[GP1:91,2] = PR[GP1:90,2] + 29.611;
   1:L PR[91] R[100]mm/sec CNT100;
   1:  PR[GP1:91,1] = PR[GP1:90,1] + -44.967;
   1:  PR[GP1:91,2] = PR[GP1:90,2] + 27.439;
   1:L PR[91] R[100]mm/sec CNT100;
   1:  PR[GP1:91,1] = PR[GP1:90,1] + -50.760;
   1:  PR[GP1:91,2] = PR[GP1:90,2] + 17.858;
   1:L PR[91] R[100]mm/sec CNT100;
   1:  PR[GP1:91,1] = PR[GP1:90,1] + -52.725;
   1:  PR[GP1:91,2] = PR[GP1:90,2] + 14.533;
   1:L PR[91] R[100]mm/sec CNT100;
   1:  PR[GP1:91,1] = PR[GP1:90,1] + -53.460;
   1:  PR[GP1:91,2] = PR[GP1:90,2] + 10.479;
   1:L PR[91] R[100]mm/sec CNT100;
   1:  PR[GP1:91,1] = PR[GP1:90,1] + -54.356;
   1:  PR[GP1:91,2] = PR[GP1:90,2] + 4.925;
   1:L PR[91] R[100]mm/sec CNT100;
   1:  PR[GP1:91,1] = PR[GP1:90,1] + -55.277;
   1:  PR[GP1:91,2] = PR[GP1:90,2] + -0.082;
   1:L PR[91] R[100]mm/sec CNT100;
   1:  PR[GP1:91,1] = PR[GP1:90,1] + -54.669;
   1:  PR[GP1:91,2] = PR[GP1:90,2] + -4.145;
   1:L PR[91] R[100]mm/sec CNT100;
   1:  PR[GP1:91,1] = PR[GP1:90,1] + -52.726;
   1:  PR[GP1:91,2] = PR[GP1:90,2] + -14.676;
   1:L PR[91] R[100]mm/sec CNT100;
   1:  PR[GP1:91,1] = PR[GP1:90,1] + -50.759;
